# B&R Automation Studio project DuctLines (part 2)

### IoMap.iom - X20CP1584/IoMap.iom
```iecst
VAR_CONFIG
	Cyclic#2.::ProcessorJogFwd AT %IX."X20DI4653a".DigitalInput01;
	Cyclic#2.::ProcessorJogRev AT %IX."X20DI4653a".DigitalInput02;
	Cyclic#1.::EStopClear AT %IX."X20DI4653a".DigitalInput04;
	Cyclic#1.::ElectricDriveEnable AT %QX."X20CM8281".DigitalOutput01;
	Cyclic#1.::ActualDAC1 AT %QW."X20CM8281".AnalogOutput01;
	Cyclic#1.::ProcessorEncoderReset AT %QX."X20DC137A".Encoder01Reset;
	Cyclic#2.::HolePunchUp AT %IX."X20DI4653".DigitalInput01;
	Cyclic#1.ProcessorDriveReady AT %IX."X20CM8281".DigitalInput01;
	Cyclic#1.CoilLineHalt AT %IX."X20DI4653".DigitalInput03;
	Cyclic#2.::PowerOn AT %IX."X20DI4653a".DigitalInput03;
	Cyclic#1.CoilLineRun AT %IX."X20DI4653".DigitalInput02;
	Cyclic#1.CoilLineReset AT %IX."X20DI4653".DigitalInput04;
	Cyclic#2.::CoilLineRunIndicator AT %QX."X20DO6639".DigitalOutput01;
	Cyclic#2.::CoilLineHaltIndicator AT %QX."X20DO6639".DigitalOutput02;
	Cyclic#2.::ShearValve AT %QX."X20DO6639".DigitalOutput04;
	Cyclic#2.LTValve AT %QX."X20DO6639a".DigitalOutput01;
	Cyclic#2.VValve AT %QX."X20DO6639a".DigitalOutput02;
	Cyclic#2.LHoleValve AT %QX."X20DO6639a".DigitalOutput03;
	Cyclic#1.LevelerBrakeSolenoid AT %QX."X20DO6639a".DigitalOutput06;
	Cyclic#2.PunchMasterShiftSolenoid AT %QX."X20DO6639b".DigitalOutput01;
	Cyclic#2.OutSideGuideSolenoid AT %QX."X20DO6639b".DigitalOutput02;
	Cyclic#2.FourFootCenterSolenoid AT %QX."X20DO6639b".DigitalOutput03;
	Cyclic#2.FiveFootCenterSolenoid AT %QX."X20DO6639b".DigitalOutput04;
	Cyclic#2.SixFootCenterSolenoid AT %QX."X20DO6639b".DigitalOutput05;
	Cyclic#2.FourFootOutsideSolenoid AT %QX."X20DO6639b".DigitalOutput06;
	Cyclic#2.FiveFootOutsideSolenoid AT %QX."X20DO6639c".DigitalOutput01;
	Cyclic#2.SixFootOutsideSolenoid AT %QX."X20DO6639c".DigitalOutput02;
	Cyclic#2.DamperHoleSolenoid AT %QX."X20DO6639c".DigitalOutput03;
	Cyclic#2.HolePunchSelectedSolenoid AT %QX."X20DO6639c".DigitalOutput04;
	Cyclic#2.DieSelectSolenoid AT %QX."X20DO6639c".DigitalOutput05;
	Cyclic#1.::ActlMetalEncoder AT %ID."X20DC137A".Encoder01;
	Cyclic#2.BackGaugeJogInPB AT %IX."X20DI4653f".DigitalInput01;
	Cyclic#2.BackGaugeJogOutPB AT %IX."X20DI4653f".DigitalInput02;
	Cyclic#2.BackGaugeHomeLS AT %IX."X20DI4653f".DigitalInput03;
	Cyclic#2.FWBResetPB AT %IX."X20DI4653f".DigitalInput04;
	Cyclic#2.::PinspotEncoderResetSignal AT %QX."X20DC137A1".Encoder01Reset;
	Cyclic#2.BrakeEncoder AT %ID."X20DC137A2".Encoder01;
	Cyclic#2.BrakeEncoderReset AT %QX."X20DC137A2".Encoder01Reset;
	Cyclic#1.::ActualDAC2 AT %QW."X20CM8281a".AnalogOutput01;
	Cyclic#2.::BrakeDriveEnable AT %QX."X20CM8281a".DigitalOutput01;
	Cyclic#2.::BrakeDriveReset AT %QX."X20CM8281a".DigitalOutput02;
	Cyclic#2.::BrakeDriveReady AT %IX."X20CM8281a".DigitalInput01;
	Cyclic#1.::TSCEF1Button AT %IX."X20DI4653c".DigitalInput01;
	Cyclic#1.::TSCEF2Button AT %IX."X20DI4653c".DigitalInput02;
	Cyclic#1.::FullCleatSelect AT %IX."X20DI4653c".DigitalInput04;
	Cyclic#2.::PartPresentPSpotter AT %IX."X20DI4653d".DigitalInput04;
	Cyclic#2.::GuideSideStopLS AT %IX."X20DI4653g".DigitalInput01;
	Cyclic#2.::OperatorSideStopLS AT %IX."X20DI4653g".DigitalInput02;
	Cyclic#2.::BrakeAutoButton AT %IX."X20DI4653g".DigitalInput03;
	Cyclic#2.::BrakeHydraulicMS AT %IX."X20DI4653g".DigitalInput04;
	Cyclic#2.LatchCylinderInLS AT %IX."X20DI4653h".DigitalInput01;
	Cyclic#2.LatchCylinderOutLS AT %IX."X20DI4653h".DigitalInput02;
	Cyclic#2.::BrakeClampUpLS AT %IX."X20DI4653h".DigitalInput03;
	Cyclic#2.::BrakeClampDownLS AT %IX."X20DI4653i".DigitalInput01;
	Cyclic#2.::FormHeadUpLS AT %IX."X20DI4653i".DigitalInput02;
	Cyclic#2.::FormHeadDownLS AT %IX."X20DI4653i".DigitalInput03;
	Cyclic#2.::RotateStopsOut AT %IX."X20DI4653i".DigitalInput04;
	Cyclic#2.::RearEjectResetLimitSwitch AT %IX."X20DI4653j".DigitalInput01;
	Cyclic#2.::SmallPartsPusherLS AT %IX."X20DI4653j".DigitalInput04;
	Cyclic#2.::ManualClampPB AT %IX."X20DI4653j".DigitalInput03;
	Cyclic#1.SlowSpeedSolenoid AT %QX."X20DO6639".DigitalOutput03;
	Cyclic#1.::ForwardFeedSolenoid AT %QX."X20DO6639a".DigitalOutput04;
	Cyclic#1.::ReverseFeedSolenoid AT %QX."X20DO6639a".DigitalOutput05;
	Cyclic#2.::PinspotterDrive AT %QX."X20DO6639g".DigitalOutput01;
	Cyclic#2.::LatchCylinderInSolenoid AT %QX."X20DO6639i".DigitalOutput01;
	Cyclic#2.::LatchCylinderOutSolenoid AT %QX."X20DO6639i".DigitalOutput02;
	Cyclic#2.::BrakeBeamRaise AT %QX."X20DO6639i".DigitalOutput03;
	Cyclic#2.::BrakeBeamLower AT %QX."X20DO6639i".DigitalOutput04;
	Cyclic#2.::BrakeStopsInSolenoid AT %QX."X20DO6639j".DigitalOutput01;
	Cyclic#2.::BrakeStopsOutSolenoid AT %QX."X20DO6639j".DigitalOutput02;
	Cyclic#2.::SideEjectSolenoid AT %QX."X20DO6639j".DigitalOutput03;
	Cyclic#2.::FormHeadDownSolenoid AT %QX."X20DO6639j".DigitalOutput04;
	Cyclic#2.SmallPartPusherFwdSolenoid AT %QX."X20DO6639k".DigitalOutput01;
	Cyclic#2.SmallPartPusherRevSolenoid AT %QX."X20DO6639k".DigitalOutput02;
	Cyclic#2.FWBUnloaderValve AT %QX."X20DO6639k".DigitalOutput03;
	Cyclic#2.BrakeAutoIndicator AT %QX."X20DO6639k".DigitalOutput04;
	Cyclic#1.::CEF1Indicator AT %QX."X20DO6639d".DigitalOutput02;
	Cyclic#1.::CEF2Indicator AT %QX."X20DO6639d".DigitalOutput03;
	Cyclic#2.::FormHeadUpSolenoid AT %QX."X20DO6639i".DigitalOutput05;
	Cyclic#2.::SideEjectLiftSolenoid AT %QX."X20DO6639i".DigitalOutput06;
	Cyclic#1.::CEFNotchDetect AT %IX."X20DC137A".DigitalInput01;
	Cyclic#2.::PinspotEncoder AT %ID."X20DC137A1".Encoder01;
	Cyclic#2.::PinspotterLoad AT %QX."X20DO6639g".DigitalOutput03;
	Cyclic#2.::LinerAirSupply AT %QX."X20DO6639g".DigitalOutput05;
	Cyclic#2.DH800TOutPB AT %IX."X20DI4653b".DigitalInput01;
	Cyclic#2.DH800TInPB AT %IX."X20DI4653b".DigitalInput02;
	Cyclic#2.DH800TOutCR AT %QX."X20DO6639e".DigitalOutput01;
	Cyclic#2.DH800TInCR AT %QX."X20DO6639e".DigitalOutput02;
	Cyclic#2.DH800CEFOutCR AT %QX."X20DO6639d".DigitalOutput01;
	Cyclic#2.DH800CEFInCR AT %QX."X20DO6639d".DigitalOutput04;
	Cyclic#2.DH800CEFCalibrateCR AT %QX."X20DO6639d".DigitalOutput05;
	Cyclic#2.DH800CEFSlowCR AT %QX."X20DO6639d".DigitalOutput06;
	Cyclic#2.::DH800CEFInPB AT %IX."X20DI4653d".DigitalInput01;
	Cyclic#2.::DH800CEFOutPB AT %IX."X20DI4653d".DigitalInput03;
	Cyclic#1.BackGaugeAirBrake AT %QX."X20DO6639k".DigitalOutput05;
	Cyclic#2.::BrakePartEjectSolenoid AT %QX."X20DO6639j".DigitalOutput05;
END_VAR
```

## Configuration E1000V2_2

### Task classes (Cpu.sw)
```
Cyclic#1 (cycle 1000 us, tolerance 0 us):
  CEF <- CEF.prg
  IMotion2 <- IMotion2.prg
  EFdrHydDrv <- EFdrHydDrv1.prg
Cyclic#2 (cycle 20000 us, tolerance 20000 us):
  SysCheck <- SysCheck.prg
  E2Feeder <- E2Feeder.prg
  PMaster <- PMaster.prg
  Pinspotter <- Pinspotter.prg
  E_FWB <- E_FWB.prg
  DH800 <- DH800.prg
Cyclic#4 (cycle 100000 us, tolerance 100000 us):
  Server <- LibAsTCP1_ST.Server.prg
Binaries: sysconf, Role, User, iomap, ashwd, asfw, arconfig, TCData
Libraries: astcp, astime, standard, asieccon, runtime, asstring
```

### Hardware
same as Physical/E1000V2_1/Hardware.hw

### IoMap.iom - X20CP1584/IoMap.iom
```iecst
VAR_CONFIG
	Cyclic#2.::ProcessorJogFwd AT %IX."X20DI4653a".DigitalInput01;
	Cyclic#2.::ProcessorJogRev AT %IX."X20DI4653a".DigitalInput02;
	Cyclic#1.::EStopClear AT %IX."X20DI4653a".DigitalInput04;
	Cyclic#1.::ElectricDriveEnable AT %QX."X20CM8281".DigitalOutput01;
	Cyclic#1.::ActualDAC1 AT %QW."X20CM8281".AnalogOutput01;
	Cyclic#1.::ProcessorEncoderReset AT %QX."X20DC137A".Encoder01Reset;
	Cyclic#2.::HolePunchUp AT %IX."X20DI4653".DigitalInput01;
	Cyclic#1.ProcessorDriveReady AT %IX."X20CM8281".DigitalInput01;
	Cyclic#1.CoilLineHalt AT %IX."X20DI4653".DigitalInput03;
	Cyclic#2.::PowerOn AT %IX."X20DI4653a".DigitalInput03;
	Cyclic#1.CoilLineRun AT %IX."X20DI4653".DigitalInput02;
	Cyclic#1.CoilLineReset AT %IX."X20DI4653".DigitalInput04;
	Cyclic#2.::CoilLineRunIndicator AT %QX."X20DO6639".DigitalOutput01;
	Cyclic#2.::CoilLineHaltIndicator AT %QX."X20DO6639".DigitalOutput02;
	Cyclic#2.::ShearValve AT %QX."X20DO6639".DigitalOutput04;
	Cyclic#2.LTValve AT %QX."X20DO6639a".DigitalOutput01;
	Cyclic#2.VValve AT %QX."X20DO6639a".DigitalOutput02;
	Cyclic#2.LHoleValve AT %QX."X20DO6639a".DigitalOutput03;
	Cyclic#1.LevelerBrakeSolenoid AT %QX."X20DO6639a".DigitalOutput06;
	Cyclic#2.PunchMasterShiftSolenoid AT %QX."X20DO6639b".DigitalOutput01;
	Cyclic#2.OutSideGuideSolenoid AT %QX."X20DO6639b".DigitalOutput02;
	Cyclic#2.FourFootCenterSolenoid AT %QX."X20DO6639b".DigitalOutput03;
	Cyclic#2.FiveFootCenterSolenoid AT %QX."X20DO6639b".DigitalOutput04;
	Cyclic#2.SixFootCenterSolenoid AT %QX."X20DO6639b".DigitalOutput05;
	Cyclic#2.FourFootOutsideSolenoid AT %QX."X20DO6639b".DigitalOutput06;
	Cyclic#2.FiveFootOutsideSolenoid AT %QX."X20DO6639c".DigitalOutput01;
	Cyclic#2.SixFootOutsideSolenoid AT %QX."X20DO6639c".DigitalOutput02;
	Cyclic#2.DamperHoleSolenoid AT %QX."X20DO6639c".DigitalOutput03;
	Cyclic#2.HolePunchSelectedSolenoid AT %QX."X20DO6639c".DigitalOutput04;
	Cyclic#2.DieSelectSolenoid AT %QX."X20DO6639c".DigitalOutput05;
	Cyclic#1.::ActlMetalEncoder AT %ID."X20DC137A".Encoder01;
	Cyclic#2.BackGaugeJogInPB AT %IX."X20DI4653f".DigitalInput01;
	Cyclic#2.BackGaugeJogOutPB AT %IX."X20DI4653f".DigitalInput02;
	Cyclic#2.BackGaugeHomeLS AT %IX."X20DI4653f".DigitalInput03;
	Cyclic#2.FWBResetPB AT %IX."X20DI4653f".DigitalInput04;
	Cyclic#2.::PinspotEncoderResetSignal AT %QX."X20DC137A1".Encoder01Reset;
	Cyclic#2.BrakeEncoder AT %ID."X20DC137A2".Encoder01;
	Cyclic#2.BrakeEncoderReset AT %QX."X20DC137A2".Encoder01Reset;
	Cyclic#1.::ActualDAC2 AT %QW."X20CM8281a".AnalogOutput01;
	Cyclic#2.::BrakeDriveEnable AT %QX."X20CM8281a".DigitalOutput01;
	Cyclic#2.::BrakeDriveReset AT %QX."X20CM8281a".DigitalOutput02;
	Cyclic#2.::BrakeDriveReady AT %IX."X20CM8281a".DigitalInput01;
	Cyclic#1.::TSCEF1Button AT %IX."X20DI4653c".DigitalInput01;
	Cyclic#1.::TSCEF2Button AT %IX."X20DI4653c".DigitalInput02;
	Cyclic#1.::FullCleatSelect AT %IX."X20DI4653c".DigitalInput04;
	Cyclic#2.::PartPresentPSpotter AT %IX."X20DI4653d".DigitalInput04;
	Cyclic#2.::GuideSideStopLS AT %IX."X20DI4653g".DigitalInput01;
	Cyclic#2.::OperatorSideStopLS AT %IX."X20DI4653g".DigitalInput02;
	Cyclic#2.::BrakeAutoButton AT %IX."X20DI4653g".DigitalInput03;
	Cyclic#2.::BrakeHydraulicMS AT %IX."X20DI4653g".DigitalInput04;
	Cyclic#2.LatchCylinderInLS AT %IX."X20DI4653h".DigitalInput01;
	Cyclic#2.LatchCylinderOutLS AT %IX."X20DI4653h".DigitalInput02;
	Cyclic#2.::BrakeClampUpLS AT %IX."X20DI4653h".DigitalInput03;
	Cyclic#2.::BrakeClampDownLS AT %IX."X20DI4653i".DigitalInput01;
	Cyclic#2.::FormHeadUpLS AT %IX."X20DI4653i".DigitalInput02;
	Cyclic#2.::FormHeadDownLS AT %IX."X20DI4653i".DigitalInput03;
	Cyclic#2.::RotateStopsOut AT %IX."X20DI4653i".DigitalInput04;
	Cyclic#2.::RearEjectResetLimitSwitch AT %IX."X20DI4653j".DigitalInput01;
	Cyclic#2.::SmallPartsPusherLS AT %IX."X20DI4653j".DigitalInput04;
	Cyclic#2.::ManualClampPB AT %IX."X20DI4653j".DigitalInput03;
	Cyclic#1.SlowSpeedSolenoid AT %QX."X20DO6639".DigitalOutput03;
	Cyclic#1.::ForwardFeedSolenoid AT %QX."X20DO6639a".DigitalOutput04;
	Cyclic#1.::ReverseFeedSolenoid AT %QX."X20DO6639a".DigitalOutput05;
	Cyclic#2.::PinspotterDrive AT %QX."X20DO6639g".DigitalOutput01;
	Cyclic#2.::LatchCylinderInSolenoid AT %QX."X20DO6639i".DigitalOutput01;
	Cyclic#2.::LatchCylinderOutSolenoid AT %QX."X20DO6639i".DigitalOutput02;
	Cyclic#2.::BrakeBeamRaise AT %QX."X20DO6639i".DigitalOutput03;
	Cyclic#2.::BrakeBeamLower AT %QX."X20DO6639i".DigitalOutput04;
	Cyclic#2.::BrakeStopsInSolenoid AT %QX."X20DO6639j".DigitalOutput01;
	Cyclic#2.::BrakeStopsOutSolenoid AT %QX."X20DO6639j".DigitalOutput02;
	Cyclic#2.::SideEjectSolenoid AT %QX."X20DO6639j".DigitalOutput03;
	Cyclic#2.::FormHeadDownSolenoid AT %QX."X20DO6639j".DigitalOutput04;
	Cyclic#2.SmallPartPusherFwdSolenoid AT %QX."X20DO6639k".DigitalOutput01;
	Cyclic#2.SmallPartPusherRevSolenoid AT %QX."X20DO6639k".DigitalOutput02;
	Cyclic#2.FWBUnloaderValve AT %QX."X20DO6639k".DigitalOutput03;
	Cyclic#2.BrakeAutoIndicator AT %QX."X20DO6639k".DigitalOutput04;
	Cyclic#1.::CEF1Indicator AT %QX."X20DO6639d".DigitalOutput02;
	Cyclic#1.::CEF2Indicator AT %QX."X20DO6639d".DigitalOutput03;
	Cyclic#2.::FormHeadUpSolenoid AT %QX."X20DO6639i".DigitalOutput05;
	Cyclic#2.::SideEjectLiftSolenoid AT %QX."X20DO6639i".DigitalOutput06;
	Cyclic#1.::CEFNotchDetect AT %IX."X20DC137A".DigitalInput01;
	Cyclic#2.::PinspotEncoder AT %ID."X20DC137A1".Encoder01;
	Cyclic#2.::PinspotterLoad AT %QX."X20DO6639g".DigitalOutput03;
	Cyclic#2.::LinerAirSupply AT %QX."X20DO6639g".DigitalOutput05;
	Cyclic#2.DH800TOutPB AT %IX."X20DI4653b".DigitalInput01;
	Cyclic#2.DH800TInPB AT %IX."X20DI4653b".DigitalInput02;
	Cyclic#2.DH800TOutCR AT %QX."X20DO6639e".DigitalOutput01;
	Cyclic#2.DH800TInCR AT %QX."X20DO6639e".DigitalOutput02;
	Cyclic#2.DH800CEFOutCR AT %QX."X20DO6639d".DigitalOutput01;
	Cyclic#2.DH800CEFInCR AT %QX."X20DO6639d".DigitalOutput04;
	Cyclic#2.DH800CEFCalibrateCR AT %QX."X20DO6639d".DigitalOutput05;
	Cyclic#2.DH800CEFSlowCR AT %QX."X20DO6639d".DigitalOutput06;
	Cyclic#2.::DH800CEFInPB AT %IX."X20DI4653d".DigitalInput01;
	Cyclic#2.::DH800CEFOutPB AT %IX."X20DI4653d".DigitalInput03;
	Cyclic#1.BackGaugeAirBrake AT %QX."X20DO6639k".DigitalOutput05;
	Cyclic#2.::BrakePartEjectSolenoid AT %QX."X20DO6639j".DigitalOutput05;
	Cyclic#2.::DH800CEFCalibratePB AT %IX."X20DI4653d".DigitalInput02;
END_VAR
```

## Configuration E2000

CPU X20CP1584, AutomationRuntime J4.25, Build 4.1.2, Vc V4.25.0, Safety 0.0

### Hardware
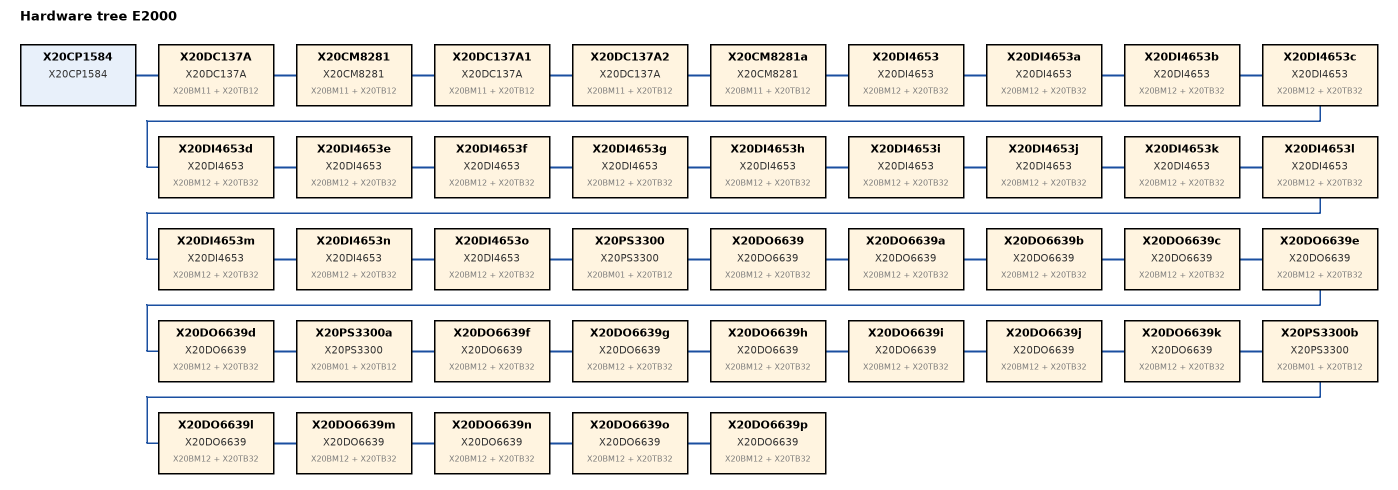
```
X20BM01 : X20BM01 v1.0.1.1  [X2X1 -> X20BM12aa.X2X2]
X20BM01a : X20BM01 v1.0.1.1  [X2X1 -> X20BM12o.X2X2]
X20BM01b : X20BM01 v1.0.1.1  [X2X1 -> X20BM12v.X2X2]
X20BM11 : X20BM11 v1.0.0.1  [X2X1 -> X20CP1584.IF6]
X20BM11a : X20BM11 v1.0.0.1  [X2X1 -> X20BM11.X2X2]
X20BM11b : X20BM11 v1.0.0.1  [X2X1 -> X20BM11a.X2X2]
X20BM11c : X20BM11 v1.0.0.1  [X2X1 -> X20BM11b.X2X2]
X20BM11d : X20BM11 v1.0.0.1  [X2X1 -> X20BM11c.X2X2]
X20BM12 : X20BM12 v1.0.0.1  [X2X1 -> X20BM11d.X2X2]
X20BM12a : X20BM12 v1.0.0.1  [X2X1 -> X20BM12.X2X2]
X20BM12aa : X20BM12 v1.0.0.1  [X2X1 -> X20BM12z.X2X2]
X20BM12ab : X20BM12 v1.0.0.1  [X2X1 -> X20BM01b.X2X2]
X20BM12ac : X20BM12 v1.0.0.1  [X2X1 -> X20BM12ab.X2X2]
X20BM12ad : X20BM12 v1.0.0.1  [X2X1 -> X20BM12ac.X2X2]
X20BM12ae : X20BM12 v1.0.0.1  [X2X1 -> X20BM12ad.X2X2]
X20BM12af : X20BM12 v1.0.0.1  [X2X1 -> X20BM12ae.X2X2]
X20BM12b : X20BM12 v1.0.0.1  [X2X1 -> X20BM12a.X2X2]
X20BM12c : X20BM12 v1.0.0.1  [X2X1 -> X20BM12b.X2X2]
X20BM12d : X20BM12 v1.0.0.1  [X2X1 -> X20BM12c.X2X2]
X20BM12e : X20BM12 v1.0.0.1  [X2X1 -> X20BM12d.X2X2]
X20BM12f : X20BM12 v1.0.0.1  [X2X1 -> X20BM12e.X2X2]
X20BM12g : X20BM12 v1.0.0.1  [X2X1 -> X20BM12f.X2X2]
X20BM12h : X20BM12 v1.0.0.1  [X2X1 -> X20BM12g.X2X2]
X20BM12i : X20BM12 v1.0.0.1  [X2X1 -> X20BM12h.X2X2]
X20BM12j : X20BM12 v1.0.0.1  [X2X1 -> X20BM12i.X2X2]
X20BM12k : X20BM12 v1.0.0.1  [X2X1 -> X20BM01.X2X2]
X20BM12l : X20BM12 v1.0.0.1  [X2X1 -> X20BM12k.X2X2]
X20BM12m : X20BM12 v1.0.0.1  [X2X1 -> X20BM12l.X2X2]
X20BM12n : X20BM12 v1.0.0.1  [X2X1 -> X20BM12m.X2X2]
X20BM12o : X20BM12 v1.0.0.1  [X2X1 -> X20BM12p.X2X2]
X20BM12p : X20BM12 v1.0.0.1  [X2X1 -> X20BM12n.X2X2]
X20BM12q : X20BM12 v1.0.0.1  [X2X1 -> X20BM01a.X2X2]
X20BM12r : X20BM12 v1.0.0.1  [X2X1 -> X20BM12q.X2X2]
X20BM12s : X20BM12 v1.0.0.1  [X2X1 -> X20BM12r.X2X2]
X20BM12t : X20BM12 v1.0.0.1  [X2X1 -> X20BM12s.X2X2]
X20BM12u : X20BM12 v1.0.0.1  [X2X1 -> X20BM12t.X2X2]
X20BM12v : X20BM12 v1.0.0.1  [X2X1 -> X20BM12u.X2X2]
X20BM12w : X20BM12 v1.0.0.1  [X2X1 -> X20BM12j.X2X2]
X20BM12x : X20BM12 v1.0.0.1  [X2X1 -> X20BM12w.X2X2]
X20BM12y : X20BM12 v1.0.0.1  [X2X1 -> X20BM12x.X2X2]
X20BM12z : X20BM12 v1.0.0.1  [X2X1 -> X20BM12y.X2X2]
X20CM8281 : X20CM8281 v1.0.4.0  [SS1 -> X20TB12a.SS; SL -> X20BM11a.SL1]
  Supervision = off
X20CM8281a : X20CM8281 v1.0.4.0  [SS1 -> X20TB12d.SS; SL -> X20BM11d.SL1]
  Supervision = off
X20CP1584 : X20CP1584 v1.3.0.0
  Connector IF2:
    ActivateDevice = 1
    EthInterfaceRedundant = 0
    Mode = Manual
    InternetAddress = 10.1.254.101
  Connector IF3:
    EplInterfaceRedundant = 0
    EplEthInterfaceRedundant = 0
  Connector IF6:
    CycleTime = 1000
  ConfigurationID = X20_CPU_E1000
  EnableUsbRemoteInstall = 1
  TimerDeviceType = EPLX2X
  TimerDevice = X20CP1584.IF6
  Cyclic1Duration = 1000
  Cyclic1Tolerance = 0
  Cyclic1Output = 1
  Cyclic2Duration = 20000
  Cyclic2Tolerance = 20000
  Cyclic3Duration = 50000
  Cyclic3Tolerance = 50000
  Cyclic4Duration = 100000
  Cyclic4Tolerance = 100000
  Cyclic5Duration = 200000
  Cyclic5Tolerance = 200000
  Cyclic6Duration = 500000
  Cyclic6Tolerance = 500000
  Cyclic7Duration = 1000000
  Cyclic7Tolerance = 1000000
  Cyclic8Duration = 10000
  Cyclic8Tolerance = 30000000
  Route1
X20DC137A : X20DC137A v1.0.0.3  [SS1 -> X20TB12.SS; SL -> X20BM11.SL1]
  Supervision = off
  CounterStd01 = 32Bit
  BWConfigChannel03 = off
X20DC137A1 : X20DC137A v1.0.0.3  [SS1 -> X20TB12b.SS; SL -> X20BM11b.SL1]
  Supervision = off
  CounterStd01 = 32Bit
  BWConfigChannel03 = off
X20DC137A2 : X20DC137A v1.0.0.3  [SS1 -> X20TB12c.SS; SL -> X20BM11c.SL1]
  Supervision = off
  CounterStd01 = 32Bit
  BWConfigChannel03 = off
X20DI4653 : X20DI4653 v1.0.2.0  [SS1 -> X20TB32.SS; SL -> X20BM12.SL1]
  Supervision = off
X20DI4653a : X20DI4653 v1.0.2.0  [SS1 -> X20TB32a.SS; SL -> X20BM12a.SL1]
  Supervision = off
X20DI4653b : X20DI4653 v1.0.2.0  [SS1 -> X20TB32b.SS; SL -> X20BM12b.SL1]
  Supervision = off
X20DI4653c : X20DI4653 v1.0.2.0  [SS1 -> X20TB32c.SS; SL -> X20BM12c.SL1]
  Supervision = off
X20DI4653d : X20DI4653 v1.0.2.0  [SS1 -> X20TB32d.SS; SL -> X20BM12d.SL1]
  Supervision = off
X20DI4653e : X20DI4653 v1.0.2.0  [SS1 -> X20TB32e.SS; SL -> X20BM12e.SL1]
  Supervision = off
X20DI4653f : X20DI4653 v1.0.2.0  [SS1 -> X20TB32f.SS; SL -> X20BM12f.SL1]
  Supervision = off
X20DI4653g : X20DI4653 v1.0.2.0  [SS1 -> X20TB32g.SS; SL -> X20BM12g.SL1]
  Supervision = off
X20DI4653h : X20DI4653 v1.0.2.0  [SS1 -> X20TB32h.SS; SL -> X20BM12h.SL1]
  Supervision = off
X20DI4653i : X20DI4653 v1.0.2.0  [SS1 -> X20TB32i.SS; SL -> X20BM12i.SL1]
  Supervision = off
X20DI4653j : X20DI4653 v1.0.2.0  [SS1 -> X20TB32j.SS; SL -> X20BM12j.SL1]
  Supervision = off
X20DI4653k : X20DI4653 v1.0.2.0  [SS1 -> X20TB32w.SS; SL -> X20BM12w.SL1]
  Supervision = off
X20DI4653l : X20DI4653 v1.0.2.0  [SS1 -> X20TB32x.SS; SL -> X20BM12x.SL1]
  Supervision = off
X20DI4653m : X20DI4653 v1.0.2.0  [SS1 -> X20TB32y.SS; SL -> X20BM12y.SL1]
  Supervision = off
X20DI4653n : X20DI4653 v1.0.2.0  [SS1 -> X20TB32z.SS; SL -> X20BM12z.SL1]
  Supervision = off
X20DI4653o : X20DI4653 v1.0.2.0  [SS1 -> X20TB32aa.SS; SL -> X20BM12aa.SL1]
  Supervision = off
X20DO6639 : X20DO6639 v1.0.1.0  [SS1 -> X20TB32k.SS; SL -> X20BM12k.SL1]
  Supervision = off
X20DO6639a : X20DO6639 v1.0.1.0  [SS1 -> X20TB32l.SS; SL -> X20BM12l.SL1]
  Supervision = off
X20DO6639b : X20DO6639 v1.0.1.0  [SS1 -> X20TB32m.SS; SL -> X20BM12m.SL1]
  Supervision = off
X20DO6639c : X20DO6639 v1.0.1.0  [SS1 -> X20TB32n.SS; SL -> X20BM12n.SL1]
  Supervision = off
X20DO6639d : X20DO6639 v1.0.1.0  [SS1 -> X20TB32o.SS; SL -> X20BM12o.SL1]
  Supervision = off
X20DO6639e : X20DO6639 v1.0.1.0  [SS1 -> X20TB32p.SS; SL -> X20BM12p.SL1]
  Supervision = off
X20DO6639f : X20DO6639 v1.0.1.0  [SS1 -> X20TB32q.SS; SL -> X20BM12q.SL1]
  Supervision = off
X20DO6639g : X20DO6639 v1.0.1.0  [SS1 -> X20TB32r.SS; SL -> X20BM12r.SL1]
  Supervision = off
X20DO6639h : X20DO6639 v1.0.1.0  [SS1 -> X20TB32s.SS; SL -> X20BM12s.SL1]
  Supervision = off
X20DO6639i : X20DO6639 v1.0.1.0  [SS1 -> X20TB32t.SS; SL -> X20BM12t.SL1]
  Supervision = off
X20DO6639j : X20DO6639 v1.0.1.0  [SS1 -> X20TB32u.SS; SL -> X20BM12u.SL1]
  Supervision = off
X20DO6639k : X20DO6639 v1.0.1.0  [SS1 -> X20TB32v.SS; SL -> X20BM12v.SL1]
  Supervision = off
X20DO6639l : X20DO6639 v1.0.1.0  [SS1 -> X20TB32ab.SS; SL -> X20BM12ab.SL1]
  Supervision = off
X20DO6639m : X20DO6639 v1.0.1.0  [SS1 -> X20TB32ac.SS; SL -> X20BM12ac.SL1]
  Supervision = off
X20DO6639n : X20DO6639 v1.0.1.0  [SS1 -> X20TB32ad.SS; SL -> X20BM12ad.SL1]
  Supervision = off
X20DO6639o : X20DO6639 v1.0.1.0  [SS1 -> X20TB32ae.SS; SL -> X20BM12ae.SL1]
  Supervision = off
X20DO6639p : X20DO6639 v1.0.1.0  [SS1 -> X20TB32af.SS; SL -> X20BM12af.SL1]
  Supervision = off
X20PS3300 : X20PS3300 v1.1.0.0  [SS1 -> X20TB12e.SS; SL -> X20BM01.SL1]
  Supervision = off
X20PS3300a : X20PS3300 v1.1.0.0  [SS1 -> X20TB12f.SS; SL -> X20BM01a.SL1]
  Supervision = off
X20PS3300b : X20PS3300 v1.1.0.0  [SS1 -> X20TB12g.SS; SL -> X20BM01b.SL1]
  Supervision = off
X20TB12 : X20TB12 v1.0.0.0
X20TB12a : X20TB12 v1.0.0.0
X20TB12b : X20TB12 v1.0.0.0
X20TB12c : X20TB12 v1.0.0.0
X20TB12d : X20TB12 v1.0.0.0
X20TB12e : X20TB12 v1.0.0.0
X20TB12f : X20TB12 v1.0.0.0
X20TB12g : X20TB12 v1.0.0.0
X20TB32 : X20TB32 v1.0.0.1
X20TB32a : X20TB32 v1.0.0.1
X20TB32aa : X20TB32 v1.0.0.1
X20TB32ab : X20TB32 v1.0.0.1
X20TB32ac : X20TB32 v1.0.0.1
X20TB32ad : X20TB32 v1.0.0.1
X20TB32ae : X20TB32 v1.0.0.1
X20TB32af : X20TB32 v1.0.0.1
X20TB32b : X20TB32 v1.0.0.1
X20TB32c : X20TB32 v1.0.0.1
X20TB32d : X20TB32 v1.0.0.1
X20TB32e : X20TB32 v1.0.0.1
X20TB32f : X20TB32 v1.0.0.1
X20TB32g : X20TB32 v1.0.0.1
X20TB32h : X20TB32 v1.0.0.1
X20TB32i : X20TB32 v1.0.0.1
X20TB32j : X20TB32 v1.0.0.1
X20TB32k : X20TB32 v1.0.0.1
X20TB32l : X20TB32 v1.0.0.1
X20TB32m : X20TB32 v1.0.0.1
X20TB32n : X20TB32 v1.0.0.1
X20TB32o : X20TB32 v1.0.0.1
X20TB32p : X20TB32 v1.0.0.1
X20TB32q : X20TB32 v1.0.0.1
X20TB32r : X20TB32 v1.0.0.1
X20TB32s : X20TB32 v1.0.0.1
X20TB32t : X20TB32 v1.0.0.1
X20TB32u : X20TB32 v1.0.0.1
X20TB32v : X20TB32 v1.0.0.1
X20TB32w : X20TB32 v1.0.0.1
X20TB32x : X20TB32 v1.0.0.1
X20TB32y : X20TB32 v1.0.0.1
X20TB32z : X20TB32 v1.0.0.1
```

### IoMap.iom - X20CP1584/IoMap.iom
```iecst
VAR_CONFIG
	Cyclic#2.Uncoiler4Select AT %IX."X20DI4653a".DigitalInput02;
	Cyclic#2.Uncoiler6Select AT %IX."X20DI4653a".DigitalInput04;
	Cyclic#1.::ElectricDriveEnable AT %QX."X20CM8281".DigitalOutput01;
	Cyclic#1.::ActualDAC1 AT %QW."X20CM8281".AnalogOutput01;
	Cyclic#1.::ProcessorEncoderReset AT %QX."X20DC137A".Encoder01Reset;
	Cyclic#2.ProcessorDriveReady AT %IX."X20CM8281".DigitalInput01;
	Cyclic#2.Uncoiler5Select AT %IX."X20DI4653a".DigitalInput03;
	Cyclic#2.::Station1ForwardSolenoid AT %QX."X20DO6639".DigitalOutput04;
	Cyclic#2.Station2ForwardSolenoid AT %QX."X20DO6639a".DigitalOutput01;
	Cyclic#2.Station2ReverseSolenoid AT %QX."X20DO6639a".DigitalOutput02;
	Cyclic#2.Station2BrakeSolenoid AT %QX."X20DO6639a".DigitalOutput03;
	Cyclic#2.Station3BrakeSolenoid AT %QX."X20DO6639a".DigitalOutput06;
	Cyclic#2.Station4ForwardSolenoid AT %QX."X20DO6639b".DigitalOutput01;
	Cyclic#2.Station4ReverseSolenoid AT %QX."X20DO6639b".DigitalOutput02;
	Cyclic#2.Station4BrakeSolenoid AT %QX."X20DO6639b".DigitalOutput03;
	Cyclic#2.Station5ForwardSolenoid AT %QX."X20DO6639b".DigitalOutput04;
	Cyclic#2.Station5ReverseSolenoid AT %QX."X20DO6639b".DigitalOutput05;
	Cyclic#2.Station5BrakeSolenoid AT %QX."X20DO6639b".DigitalOutput06;
	Cyclic#2.Station6ForwardSolenoid AT %QX."X20DO6639c".DigitalOutput01;
	Cyclic#2.Station6ReverseSolenoid AT %QX."X20DO6639c".DigitalOutput02;
	Cyclic#2.Station6BrakeSolenoid AT %QX."X20DO6639c".DigitalOutput03;
	Cyclic#1.::ActlMetalEncoder AT %ID."X20DC137A".Encoder01;
	Cyclic#2.PinspotEncoder AT %ID."X20DC137A1".Encoder01;
	Cyclic#2.PinspotEncoderResetSignal AT %QX."X20DC137A1".Encoder01Reset;
	Cyclic#1.BrakeEncoder AT %ID."X20DC137A2".Encoder01;
	Cyclic#1.BrakeDriveEnable AT %QX."X20CM8281a".DigitalOutput01;
	Cyclic#1.BrakeDriveReset AT %QX."X20CM8281a".DigitalOutput02;
	Cyclic#2.BrakeDriveReady AT %IX."X20CM8281a".DigitalInput01;
	Cyclic#2.UncoilerAutoSwitch AT %IX."X20DI4653".DigitalInput01;
	Cyclic#2.UncoilerJogPB AT %IX."X20DI4653".DigitalInput02;
	Cyclic#2.Uncoiler1Select AT %IX."X20DI4653".DigitalInput03;
	Cyclic#2.Uncoiler2Select AT %IX."X20DI4653".DigitalInput04;
	Cyclic#2.Uncoiler3Select AT %IX."X20DI4653a".DigitalInput01;
	Cyclic#2.UncoilerStationLimitSwitch1 AT %IX."X20DI4653b".DigitalInput01;
	Cyclic#2.UncoilerStationLimitSwitch2 AT %IX."X20DI4653b".DigitalInput02;
	Cyclic#2.UncoilerStationLimitSwitch3 AT %IX."X20DI4653b".DigitalInput03;
	Cyclic#2.UncoilerStationLimitSwitch4 AT %IX."X20DI4653b".DigitalInput04;
	Cyclic#2.UncoilerStationLimitSwitch5 AT %IX."X20DI4653c".DigitalInput01;
	Cyclic#2.UncoilerStationLimitSwitch6 AT %IX."X20DI4653c".DigitalInput02;
	Cyclic#2.UncoilerRewindSwitch AT %IX."X20DI4653c".DigitalInput03;
	Cyclic#2.UncoilerUnwindSwitch AT %IX."X20DI4653c".DigitalInput04;
	Cyclic#2.HolePunchUp AT %IX."X20DI4653d".DigitalInput01;
	Cyclic#2.::ProcessorJogFwd AT %IX."X20DI4653d".DigitalInput02;
	Cyclic#2.::ProcessorJogRev AT %IX."X20DI4653d".DigitalInput03;
	Cyclic#1.PowerOn AT %IX."X20DI4653e".DigitalInput02;
	Cyclic#1.EStopClear AT %IX."X20DI4653e".DigitalInput04;
	Cyclic#2.HeadInPositionLS AT %IX."X20DI4653f".DigitalInput01;
	Cyclic#2.Pusher1OffProx AT %IX."X20DI4653f".DigitalInput02;
	Cyclic#2.Pusher2OffProx AT %IX."X20DI4653f".DigitalInput03;
	Cyclic#2.Table1SheetStopProxA AT %IX."X20DI4653f".DigitalInput04;
	Cyclic#2.Table1SheetStopProxB AT %IX."X20DI4653g".DigitalInput01;
	Cyclic#2.Table2SheetStopProxA AT %IX."X20DI4653g".DigitalInput02;
	Cyclic#2.Table2SheetStopProxB AT %IX."X20DI4653g".DigitalInput03;
	Cyclic#2.Lift3DownProx AT %IX."X20DI4653g".DigitalInput04;
	Cyclic#2.BypassSwitch AT %IX."X20DI4653h".DigitalInput01;
	Cyclic#2.Table1SideBypassLS AT %IX."X20DI4653h".DigitalInput02;
	Cyclic#2.CEFJogPB AT %IX."X20DI4653h".DigitalInput04;
	Cyclic#2.TDFJogPB AT %IX."X20DI4653i".DigitalInput01;
	Cyclic#2.LOMSpeedSelect1 AT %IX."X20DI4653i".DigitalInput02;
	Cyclic#2.LOMSpeedSelect2 AT %IX."X20DI4653i".DigitalInput03;
	Cyclic#2.::PartPresentPSpotter AT %IX."X20DI4653i".DigitalInput04;
	Cyclic#2.GuideSideStopLS AT %IX."X20DI4653j".DigitalInput01;
	Cyclic#2.OperatorSideStopLS AT %IX."X20DI4653j".DigitalInput02;
	Cyclic#2.BrakeClampUpLS AT %IX."X20DI4653j".DigitalInput03;
	Cyclic#2.BrakeClampMidwayLS AT %IX."X20DI4653j".DigitalInput04;
	Cyclic#2.BrakeClampDownLS AT %IX."X20DI4653k".DigitalInput01;
	Cyclic#2.FormHeadUpLS AT %IX."X20DI4653k".DigitalInput02;
	Cyclic#2.FormHeadDownLS AT %IX."X20DI4653k".DigitalInput03;
	Cyclic#2.RearEjectResetLimitSwitch AT %IX."X20DI4653k".DigitalInput04;
	Cyclic#2.BackGaugeHomeLS AT %IX."X20DI4653l".DigitalInput01;
	Cyclic#2.ManualClampPB AT %IX."X20DI4653l".DigitalInput02;
	Cyclic#2.SmallPartsPusherLS AT %IX."X20DI4653l".DigitalInput03;
	Cyclic#2.BackGaugeJogInPB AT %IX."X20DI4653l".DigitalInput04;
	Cyclic#2.BackGaugeJogOutPB AT %IX."X20DI4653m".DigitalInput01;
	Cyclic#2.SmallPartPusherHomeLS AT %IX."X20DI4653m".DigitalInput02;
	Cyclic#2.PartEjectHomeLS AT %IX."X20DI4653m".DigitalInput03;
	Cyclic#2.TripIndicatorCradles2 AT %IX."X20DI4653n".DigitalInput01;
	Cyclic#2.TripIndicatorCoilLine AT %IX."X20DI4653n".DigitalInput02;
	Cyclic#2.TripIndicatorTransfer1 AT %IX."X20DI4653n".DigitalInput03;
	Cyclic#2.TripIndicatorTransfer2 AT %IX."X20DI4653n".DigitalInput04;
	TripIndicatorCEF AT %IX."X20DI4653o".DigitalInput01;
	TripIndicatorTDF AT %IX."X20DI4653o".DigitalInput02;
	TripIndicatorPump AT %IX."X20DI4653o".DigitalInput03;
	Cyclic#2.BrakeHydraulics AT %IX."X20DI4653o".DigitalInput04;
	Cyclic#2.::Station1ReverseSolenoid AT %QX."X20DO6639".DigitalOutput05;
	Cyclic#2.::Station1BrakeSolenoid AT %QX."X20DO6639".DigitalOutput06;
	Cyclic#2.Statrion3ForwardSolenoid AT %QX."X20DO6639a".DigitalOutput04;
	Cyclic#2.Station3ReverseSolenoid AT %QX."X20DO6639a".DigitalOutput05;
	Cyclic#2.::FourFootCenterSolenoid AT %QX."X20DO6639e".DigitalOutput02;
	Cyclic#2.::LHoleValve AT %QX."X20DO6639e".DigitalOutput01;
	Cyclic#2.FiveFootCenterSolenoid AT %QX."X20DO6639e".DigitalOutput03;
	Cyclic#2.SixFootCenterSolenoid AT %QX."X20DO6639e".DigitalOutput04;
	Cyclic#2.::FourFootOutsideSolenoid AT %QX."X20DO6639d".DigitalOutput01;
	Cyclic#2.::FiveFootOutsideSolenoid AT %QX."X20DO6639d".DigitalOutput02;
	Cyclic#2.::SixFootOutsideSolenoid AT %QX."X20DO6639d".DigitalOutput03;
	Cyclic#2.::OutSideGuideSolenoid AT %QX."X20DO6639d".DigitalOutput04;
	Cyclic#2.::PunchMasterShiftSolenoid AT %QX."X20DO6639f".DigitalOutput01;
	Cyclic#2.DamperHoleSolenoid AT %QX."X20DO6639f".DigitalOutput02;
	Cyclic#1.SlowSpeedSolenoid AT %QX."X20DO6639f".DigitalOutput03;
	Cyclic#1.ForwardFeedSolenoid AT %QX."X20DO6639f".DigitalOutput04;
	Cyclic#1.ReverseFeedSolenoid AT %QX."X20DO6639f".DigitalOutput05;
	Cyclic#1.LevelerBrakeSolenoid AT %QX."X20DO6639f".DigitalOutput06;
	Cyclic#2.::ShearValve AT %QX."X20DO6639g".DigitalOutput01;
	Cyclic#2.::LTValve AT %QX."X20DO6639g".DigitalOutput02;
	Cyclic#2.::VValve AT %QX."X20DO6639g".DigitalOutput03;
	Cyclic#2.CoilLinePower AT %QX."X20DO6639g".DigitalOutput04;
	Cyclic#2.EZPunchSolenoid AT %QX."X20DO6639g".DigitalOutput05;
	Cyclic#2.Transfer1Power AT %QX."X20DO6639h".DigitalOutput01;
	Cyclic#2.Transfer2Power AT %QX."X20DO6639h".DigitalOutput02;
	Cyclic#2.Lift1Solenoid AT %QX."X20DO6639h".DigitalOutput03;
	Cyclic#2.Lift2Solenoid AT %QX."X20DO6639h".DigitalOutput04;
	Cyclic#2.Lift3UpSolenoid AT %QX."X20DO6639i".DigitalOutput01;
	Cyclic#2.Lift3DownSolenoid AT %QX."X20DO6639i".DigitalOutput02;
	Cyclic#2.Pusher1Solenoid AT %QX."X20DO6639i".DigitalOutput03;
	Cyclic#2.Pusher2Solenoid AT %QX."X20DO6639i".DigitalOutput04;
	Cyclic#1.StatHeadRollSolenoid AT %QX."X20DO6639j".DigitalOutput01;
	Cyclic#1.MoveHeadRollSolenoid AT %QX."X20DO6639j".DigitalOutput02;
	Cyclic#2.CEFPower AT %QX."X20DO6639j".DigitalOutput03;
	TDFPower AT %QX."X20DO6639k".DigitalOutput01;
	Cyclic#2.LOMLowSpeedRelay AT %QX."X20DO6639l".DigitalOutput01;
	Cyclic#2.LOMHiSpeedRelay AT %QX."X20DO6639l".DigitalOutput02;
	Cyclic#2.BrakeLowSpeedRelay AT %QX."X20DO6639l".DigitalOutput03;
	Cyclic#2.BrakeHiSpeedRelay AT %QX."X20DO6639l".DigitalOutput04;
	Cyclic#2.::PinspotterDrive AT %QX."X20DO6639m".DigitalOutput01;
	Cyclic#2.LOMConveyorRunRelay AT %QX."X20DO6639m".DigitalOutput02;
	Cyclic#2.::PinspotterLoad AT %QX."X20DO6639m".DigitalOutput03;
	Cyclic#2.LinerAirSupply AT %QX."X20DO6639m".DigitalOutput04;
	Cyclic#2.BrakeHydraulicMS AT %QX."X20DO6639n".DigitalOutput01;
	Cyclic#2.BrakeOutfeedConveyorMotor AT %QX."X20DO6639n".DigitalOutput02;
	Cyclic#2.::BrakeBeamRaise AT %QX."X20DO6639n".DigitalOutput03;
	Cyclic#2.::BrakeBeamLower AT %QX."X20DO6639n".DigitalOutput04;
	Cyclic#2.FormHeadUpSolenoid AT %QX."X20DO6639o".DigitalOutput01;
	Cyclic#2.BrakeStopsInSolenoid AT %QX."X20DO6639o".DigitalOutput02;
	Cyclic#2.BrakeStopsOutSolenoid AT %QX."X20DO6639o".DigitalOutput03;
	Cyclic#2.BrakePartEjectSolenoid AT %QX."X20DO6639o".DigitalOutput04;
	Cyclic#2.SmallPartPusherFwdSolenoid AT %QX."X20DO6639p".DigitalOutput01;
	Cyclic#2.SmallPartPusherRevSolenoid AT %QX."X20DO6639p".DigitalOutput02;
	Cyclic#1.BackGaugeAirBrake AT %QX."X20DO6639p".DigitalOutput03;
	Cyclic#2.BrakeInfeedConveyorMotor AT %QX."X20DO6639p".DigitalOutput04;
	Cyclic#2.::BrakeEncoderReset AT %QX."X20DC137A2".Encoder01Reset;
	Cyclic#2.CDADecoilPower AT %QX."X20DO6639".DigitalOutput01;
	Cyclic#1.::CEFNotchDetect AT %IX."X20DC137A".DigitalInput01;
	Cyclic#1.::ActualDAC2 AT %QW."X20CM8281a".AnalogOutput01;
END_VAR
```

## Configuration Southwark_CD2505_00

### Task classes (Cpu.sw)
```
Cyclic#1 (cycle 1000 us, tolerance 10000 us):
  IMotionCon <- IMotionControl.prg
  CleatRoll <- CleatRoll.prg
Cyclic#2 (cycle 10000 us, tolerance 20000 us):
  Uncoiler_1 <- Uncoiler_1.prg
  MarkTable <- MarkTable.prg
  MarkRF <- MarkRF.prg
  Feeder <- Feeder.prg
  SBrake <- SBrake.prg
  Pivot_2 <- Pivot_2.prg
  TDCTable <- TDCTable.prg
  TDCRFPshrs <- TDCRFPshrs.prg
  GlueApp <- GlueApp.prg
  Insulmatic <- Insulmatic.prg
  Pinspotter <- Pinspotter.prg
  BrakeCommo <- BrakeCommon.prg
  HydraulicB <- HydraulicBrakeCarriage.prg
  HWBwoPLC <- HWBwoPLC.prg
Cyclic#4 (cycle 100000 us, tolerance 100000 us):
  HMIButtons <- HMIButtons.prg
  Server <- LibAsTCP1_ST.Server.prg
Binaries: TCData, arconfig, asfw, ashwd, iomap, User, Role, sysconf
Libraries: standard, MestekLib, AsTCP, runtime, asstring, asieccon, astime
```

### Hardware
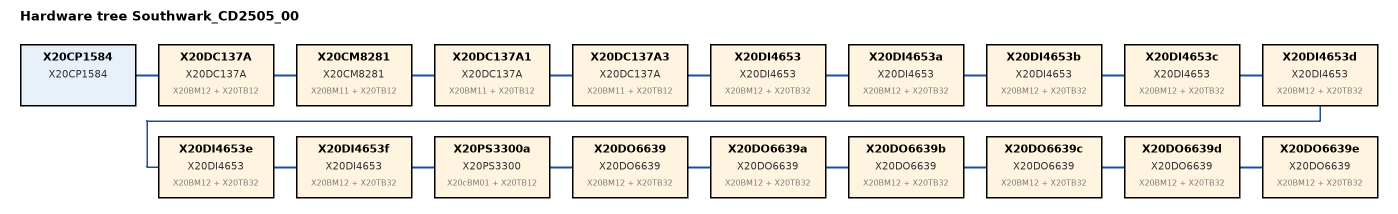
```
X20BM11 : X20BM11 v1.0.0.1  [X2X1 -> X20BM12a.X2X2]
X20BM11b : X20BM11 v1.0.0.1  [X2X1 -> X20BM11.X2X2]
X20BM11c : X20BM11 v1.0.0.1  [X2X1 -> X20BM11b.X2X2]
X20BM12 : X20BM12 v1.0.0.1  [X2X1 -> X20BM11c.X2X2]
X20BM12a : X20BM12 v1.0.0.1  [X2X1 -> X20CP1584.IF6]
X20BM12aa : X20BM12 v1.0.0.1  [X2X1 -> X20BM12z.X2X2]
X20BM12b : X20BM12 v1.0.0.1  [X2X1 -> X20BM12.X2X2]
X20BM12c : X20BM12 v1.0.0.1  [X2X1 -> X20BM12b.X2X2]
X20BM12d : X20BM12 v1.0.0.1  [X2X1 -> X20BM12c.X2X2]
X20BM12e : X20BM12 v1.0.0.1  [X2X1 -> X20BM12d.X2X2]
X20BM12f : X20BM12 v1.0.0.1  [X2X1 -> X20BM12e.X2X2]
X20BM12g : X20BM12 v1.0.0.1  [X2X1 -> X20BM12f.X2X2]
X20BM12v : X20BM12 v1.0.0.1  [X2X1 -> X20cBM01.X2X2]
X20BM12w : X20BM12 v1.0.0.1  [X2X1 -> X20BM12v.X2X2]
X20BM12x : X20BM12 v1.0.0.1  [X2X1 -> X20BM12w.X2X2]
X20BM12y : X20BM12 v1.0.0.1  [X2X1 -> X20BM12x.X2X2]
X20BM12z : X20BM12 v1.0.0.1  [X2X1 -> X20BM12y.X2X2]
X20CM8281 : X20CM8281 v1.0.4.0  [SS1 -> X20TB12.SS; SL -> X20BM11.SL1]
  Supervision = off
X20CP1584 : X20CP1584 v1.3.0.0
  Connector IF2:
    ActivateDevice = 1
    EthInterfaceRedundant = 0
    Mode = Manual
    InternetAddress = 10.1.254.101
  Connector IF3:
    EplInterfaceRedundant = 0
    EplEthInterfaceRedundant = 0
  ConfigurationID = X20_CPU_test
  EnableUsbRemoteInstall = 1
  TimerDeviceType = SWIOTIMER
  Cyclic1Duration = 1000
  Cyclic1Tolerance = 10000
  Cyclic2Duration = 10000
  Cyclic2Tolerance = 20000
  Cyclic3Duration = 50000
  Cyclic3Tolerance = 50000
  Cyclic4Duration = 100000
  Cyclic4Tolerance = 100000
  Cyclic5Duration = 200000
  Cyclic5Tolerance = 200000
  Cyclic6Duration = 500000
  Cyclic6Tolerance = 500000
  Cyclic7Duration = 1000000
  Cyclic7Tolerance = 1000000
  Cyclic8Duration = 10000
  Cyclic8Tolerance = 30000000
X20DC137A : X20DC137A v1.0.0.3  [SS1 -> X20TB12b.SS; SL -> X20BM12a.SL1]
  Supervision = off
  CounterStd01 = 32Bit
  BWConfigChannel03 = off
X20DC137A1 : X20DC137A v1.0.0.3  [SS1 -> X20TB12c.SS; SL -> X20BM11b.SL1]
  Supervision = off
  CounterStd01 = 32Bit
  BWConfigChannel03 = off
X20DC137A3 : X20DC137A v1.0.0.3  [SS1 -> X20TB12d.SS; SL -> X20BM11c.SL1]
  Supervision = off
  CounterStd01 = 32Bit
  BWConfigChannel03 = off
X20DI4653 : X20DI4653 v1.0.2.0  [SS1 -> X20TB32.SS; SL -> X20BM12.SL1]
  Supervision = off
X20DI4653a : X20DI4653 v1.0.2.0  [SS1 -> X20TB32a.SS; SL -> X20BM12b.SL1]
  Supervision = off
X20DI4653b : X20DI4653 v1.0.2.0  [SS1 -> X20TB32b.SS; SL -> X20BM12c.SL1]
  Supervision = off
X20DI4653c : X20DI4653 v1.0.2.0  [SS1 -> X20TB32c.SS; SL -> X20BM12d.SL1]
  Supervision = off
X20DI4653d : X20DI4653 v1.0.2.0  [SS1 -> X20TB32d.SS; SL -> X20BM12e.SL1]
  Supervision = off
X20DI4653e : X20DI4653 v1.0.2.0  [SS1 -> X20TB32e.SS; SL -> X20BM12f.SL1]
  Supervision = off
X20DI4653f : X20DI4653 v1.0.2.0  [SS1 -> X20TB32f.SS; SL -> X20BM12g.SL1]
  Supervision = off
X20DO6639 : X20DO6639 v1.0.1.0  [SS1 -> X20TB32u.SS; SL -> X20BM12v.SL1]
  Supervision = off
X20DO6639a : X20DO6639 v1.0.1.0  [SS1 -> X20TB32v.SS; SL -> X20BM12w.SL1]
  Supervision = off
X20DO6639b : X20DO6639 v1.0.1.0  [SS1 -> X20TB32w.SS; SL -> X20BM12x.SL1]
  Supervision = off
X20DO6639c : X20DO6639 v1.0.1.0  [SS1 -> X20TB32x.SS; SL -> X20BM12y.SL1]
  Supervision = off
X20DO6639d : X20DO6639 v1.0.1.0  [SS1 -> X20TB32y.SS; SL -> X20BM12z.SL1]
  Supervision = off
X20DO6639e : X20DO6639 v1.0.1.0  [SS1 -> X20TB32z.SS; SL -> X20BM12aa.SL1]
  Supervision = off
X20PS3300a : X20PS3300 v1.1.0.0  [SS1 -> X20TB12f.SS; SL -> X20cBM01.SL1]
  Supervision = off
X20TB12 : X20TB12 v1.0.0.0
X20TB12b : X20TB12 v1.0.0.0
X20TB12c : X20TB12 v1.0.0.0
X20TB12d : X20TB12 v1.0.0.0
X20TB12f : X20TB12 v1.0.0.0
X20TB32 : X20TB32 v1.0.0.1
X20TB32a : X20TB32 v1.0.0.1
X20TB32b : X20TB32 v1.0.0.1
X20TB32c : X20TB32 v1.0.0.1
X20TB32d : X20TB32 v1.0.0.1
X20TB32e : X20TB32 v1.0.0.1
X20TB32f : X20TB32 v1.0.0.1
X20TB32u : X20TB32 v1.0.0.1
X20TB32v : X20TB32 v1.0.0.1
X20TB32w : X20TB32 v1.0.0.1
X20TB32x : X20TB32 v1.0.0.1
X20TB32y : X20TB32 v1.0.0.1
X20TB32z : X20TB32 v1.0.0.1
X20cBM01 : X20cBM01 v1.0.1.0  [X2X1 -> X20BM12g.X2X2]
```

### IoMap.iom - X20CP1584/IoMap.iom
```iecst
VAR_CONFIG
	Cyclic#1.ActlMetalEncoder AT %ID."X20DC137A".Encoder01;
	Cyclic#1.::ProcessorEncoderReset AT %QX."X20DC137A".Encoder01Reset;
	Cyclic#1.ActualDAC1 AT %QW."X20CM8281".AnalogOutput01;
	Cyclic#1.ElectricDriveEnable AT %QX."X20CM8281".DigitalOutput01;
	Cyclic#2.MarkEncoderResetSignal AT %QX."X20DC137A1".Encoder01Reset;
	Cyclic#2.RawMarkEncoder AT %ID."X20DC137A1".Encoder01;
	Cyclic#2.::BrakeEncoderReset AT %QX."X20DC137A3".Encoder01Reset;
	Cyclic#2.BrakeEncoder AT %ID."X20DC137A3".Encoder01;
	Cyclic#2.EStopClear AT %IX."X20DI4653".DigitalInput01;
	Cyclic#2.FeedInitButton AT %IX."X20DI4653".DigitalInput04;
	Cyclic#2.ProcessorDriveEnable AT %IX."X20DI4653".DigitalInput03;
	Cyclic#2.UncoilerOnLatch AT %IX."X20DI4653".DigitalInput02;
	Cyclic#2.DuctoAuto AT %IX."X20DI4653a".DigitalInput01;
	Cyclic#2.MatlAtMeasureRoll AT %IX."X20DI4653a".DigitalInput04;
	Cyclic#2.ProcessorJogFwd AT %IX."X20DI4653a".DigitalInput02;
	Cyclic#2.ProcessorJogRev AT %IX."X20DI4653a".DigitalInput03;
	Cyclic#2.RotatingTableOn AT %IX."X20DI4653b".DigitalInput01;
	Cyclic#2.PartPresentRTClamp AT %IX."X20DI4653b".DigitalInput02;
	Cyclic#2.PartPresentRTKnurledRoll AT %IX."X20DI4653b".DigitalInput03;
	Cyclic#2.PartRotateComplete AT %IX."X20DI4653b".DigitalInput04;
	Cyclic#2.HumpLimitSwitch AT %IX."X20DI4653c".DigitalInput01;
	Cyclic#2.PowerOn AT %IX."X20DI4653c".DigitalInput04;
	Cyclic#2.SlackBar AT %IX."X20DI4653c".DigitalInput02;
	Cyclic#2.MarkAuto AT %IX."X20DI4653d".DigitalInput02;
	Cyclic#2.MarkRollformerOn AT %IX."X20DI4653d".DigitalInput01;
	Cyclic#2.MarkSetButton AT %IX."X20DI4653d".DigitalInput03;
	Cyclic#2.::MarkRefSwitch AT %IX."X20DI4653e".DigitalInput01;
	Cyclic#2.MarkHeadJogInSwitch AT %IX."X20DI4653e".DigitalInput03;
	Cyclic#2.MarkHeadJogOutSwitch AT %IX."X20DI4653e".DigitalInput04;
	Cyclic#2.MarkHiSpeedSignal AT %IX."X20DI4653e".DigitalInput02;
	Cyclic#2.::CarriageReference AT %IX."X20DI4653f".DigitalInput01;
	Cyclic#2.::BrakeAutoRequest AT %IX."X20DI4653f".DigitalInput03;
	Cyclic#2.AmberLight AT %QX."X20DO6639".DigitalOutput02;
	Cyclic#2.BatchActivePhysical AT %QX."X20DO6639".DigitalOutput06;
	Cyclic#2.BlockingValve AT %QX."X20DO6639".DigitalOutput05;
	Cyclic#2.BlueLight AT %QX."X20DO6639".DigitalOutput03;
	Cyclic#2.UncoilerRun AT %QX."X20DO6639".DigitalOutput04;
	Cyclic#2.WarningHorn AT %QX."X20DO6639".DigitalOutput01;
	Cyclic#2.LTValve AT %QX."X20DO6639a".DigitalOutput04;
	Cyclic#2.::CustomVValve AT %QX."X20DO6639a".DigitalOutput06;
	Cyclic#2.::CustomLTValve AT %QX."X20DO6639a".DigitalOutput05;
	Cyclic#2.ShearValve AT %QX."X20DO6639a".DigitalOutput01;
	Cyclic#2.SnapLockButtonGag AT %QX."X20DO6639a".DigitalOutput02;
	Cyclic#2.VValve AT %QX."X20DO6639a".DigitalOutput03;
	Cyclic#2.RTSkewTableRelay AT %QX."X20DO6639b".DigitalOutput01;
	Cyclic#2.RTBeltConveyorMotor AT %QX."X20DO6639b".DigitalOutput02;
	Cyclic#2.RTKnurledRollsMotor AT %QX."X20DO6639b".DigitalOutput03;
	Cyclic#2.RTBeltConveyorRaiseSolenoid AT %QX."X20DO6639b".DigitalOutput04;
	Cyclic#2.PivotClampCloseSolenoid AT %QX."X20DO6639b".DigitalOutput05;
	Cyclic#2.CushionRollRaiseSolenoid AT %QX."X20DO6639b".DigitalOutput06;
	Cyclic#2.RTPivotArmRotate AT %QX."X20DO6639c".DigitalOutput03;
	Cyclic#2.RTKnurledRollLowerSolenoid AT %QX."X20DO6639c".DigitalOutput01;
	Cyclic#2.RTKnurledRollGateSolenoid AT %QX."X20DO6639c".DigitalOutput02;
	Cyclic#2.::MarkRFHighSpeed AT %QX."X20DO6639d".DigitalOutput03;
	Cyclic#2.::BrakeHighSpeedRelay AT %QX."X20DO6639e".DigitalOutput03;
	Cyclic#2.::BrakeOn AT %QX."X20DO6639e".DigitalOutput04;
	::PartPresentMarkExit AT %IX."X20DI4653c".DigitalInput03;
	Cyclic#2.SmallPittsSelected AT %IX."X20DI4653d".DigitalInput04;
	Cyclic#2.::MarkRFMoveIn AT %QX."X20DO6639d".DigitalOutput01;
	Cyclic#2.::BrakeSetButton AT %IX."X20DI4653f".DigitalInput02;
	Cyclic#2.::MarkRFMoveOut AT %QX."X20DO6639d".DigitalOutput02;
	Cyclic#2.Brake8Inch2ndLeg AT %QX."X20DO6639e".DigitalOutput05;
	Cyclic#2.::MoveToBeam AT %QX."X20DO6639e".DigitalOutput01;
	Cyclic#2.::MoveAwayBeam AT %QX."X20DO6639e".DigitalOutput02;
END_VAR
```

## Configuration sim

CPU PC_any, AutomationRuntime J4.25, Build 4.1.2, Vc V4.25.0, Safety 0.0

### Task classes (Cpu.sw)
```
Cyclic#1 (cycle 10000 us, tolerance 10000 us):
  Server <- LibAsTCP1_ST.Server.prg
  MotionCont <- MotionControl1.prg
Cyclic#2 (cycle 20000 us, tolerance 50000000 us):
  Feeder <- Feeder.prg
  MarkTable <- MarkTable.prg
  MarkRF <- MarkRF.prg
  TDCTable <- TDCTable.prg
  TDCRFPshrs <- TDCRFPshrs.prg
  Insulmatic <- Insulmatic.prg
  GlueApp <- GlueApp.prg
  Pinspotter <- Pinspotter.prg
  BrakeCommo <- BrakeCommon.prg
  HWBwoPLC <- HWBwoPLC.prg
  HydraulicB <- HydraulicBrakeCarriage.prg
  CleatRoll <- CleatRoll.prg
Cyclic#4 (cycle 100000 us, tolerance 10000000 us):
  HMIButtons <- HMIButtons.prg
Cyclic#5 (cycle 2000000 us, tolerance 10000000 us):
  LampTest <- LampTest.prg
  Client <- LibAsTCP1_ST.Client.prg
Binaries: TCData, arconfig, asfw, ashwd, iomap, User, Role, sysconf
Libraries: standard, MestekLib, runtime, asieccon, astime, Library, asstring, astcp
```

### Hardware
```
PC : PC_any v1.1.0.0 (OrderNumber=PC)
  Connector IF1:
    ActivateDevice = 1
    ActivateIna = 1
  Connector IF3:
    InaPort = 11159
  ConfigurationID = X20_CPU_Config1
  Cyclic1Duration = 10000
  Cyclic1Tolerance = 10000
  Cyclic2Duration = 20000
  Cyclic2Tolerance = 50000000
  Cyclic3Duration = 50000
  Cyclic3Tolerance = 10000000
  Cyclic4Duration = 100000
  Cyclic4Tolerance = 10000000
  Cyclic5Duration = 2000000
  Cyclic5Tolerance = 10000000
  Cyclic6Duration = 3000000
  Cyclic6Tolerance = 12000000
  Cyclic7Duration = 4000000
  Cyclic7Tolerance = 12000000
  Cyclic8Duration = 5000000
  Cyclic8Tolerance = 30000000
```

## Logical view

Binary libraries used (declarations not repeated): operator, runtime, astime, AsIecCon, standard, AsTCP, asstring

### Global.var - Global variables
```iecst
VAR
	AccelRampReal : REAL := 500.0;
	AccelRampReal2 : REAL := 1000.0;
	ActlMetalEncoder : DINT;
	ActualDAC1 : INT;
	ActualDAC2 : INT;
	ActualMetalPosition : REAL; (*Scaled Material Position*)
	ActualRunPercent : REAL;
	ActualSpeed1 : REAL; (*Inches Per Second*)
	AdjustableTDCHeadActual : REAL;
	AdjustableTDCHeadDesired : REAL;
	AdjustableTDCHeadReference : REAL;
	AllSystemsOK : BOOL;
	AmberLight : BOOL;
	Analog1Forward : BOOL;
	Analog1Reverse : BOOL;
	AverageSpeed1 : REAL;
	BackGaugeAirBrake : BOOL;
	BackGaugeHomeLS : BOOL;
	BackGaugeJogInPB : BOOL;
	BackGaugeJogOutPB : BOOL;
	BackGaugeJogPercent : DINT;
	BackGaugeRunPercent : DINT;
	BatchActivePhysical : BOOL;
	BatchCancelSignal : BOOL;
	BC_Home4 : BOOL;
	BDelay1 : DINT;
	BDelay2 : DINT;
	BeadRollHits : DINT;
	BeadRollIndex : UINT;
	BeadRollJob : DINT;
	BeadRollMove : REAL;
	BeadRollTable : ARRAY[0..9] OF REAL;
	BeginEjectStep : BOOL;
	BeginMarkHoming : BOOL;
	BendingAgain : BOOL;
	BendingLatch : BOOL;
	BendInProcess : BOOL;
	BendSequenceReset : BOOL;
	BendStart : BOOL;
	BlockingValve : BOOL;
	BlockingValveButton : BOOL;
	BlueLight : BOOL;
	Brake8Inch2ndLeg : BOOL;
	BrakeActive : BOOL;
	BrakeActual : REAL := 20.0;
	BrakeArmLwrInhibit : BOOL;
	BrakeAuto : BOOL;
	BrakeAutoButton : BOOL;
	BrakeAutoIndicator : BOOL;
	BrakeAutoRequest : BOOL;
	BrakeBeamDownProx : BOOL;
	BrakeBeamLower : BOOL;
	BrakeBeamLwrInhibit : BOOL;
	BrakeBeamRaise : BOOL;
	BrakeBeamUpProx : BOOL;
	BrakeCarriageHomePosition : REAL;
	diBrakeCarriageJogIn : BOOL;
	diBrakeCarriageJogOut : BOOL;
	BrakeCarriageTarget : REAL;
	BrakeClampDownLS : BOOL;
	BrakeClampMidwayLS : BOOL;
	BrakeClampUpLS : BOOL;
	BrakeConveyorHigh : BOOL;
	BrakeConveyorLow : BOOL;
	BrakeDesired : REAL := 20.0;
	BrakeDriveEnable : BOOL;
	BrakeDriveFaultReset : BOOL;
	BrakeDriveReady : BOOL;
	BrakeDriveReset : BOOL;
	BrakeEncoder : DINT;
	BrakeEncoderReset : BOOL;
	BrakeHighSpeedRelay : BOOL;
	BrakeHiSpeedRelay : BOOL;
	BrakeHydraulicMS : BOOL;
	BrakeHydraulics : BOOL;
	BrakeIGain : DINT;
	BrakeInfeedConveyorMotor : BOOL;
	BrakeIsRefed : BOOL;
	BrakeIsSetUp : BOOL;
	BrakeJob : DINT;
	BrakeLeafHomeProx : BOOL;
	BrakeLeafLower : BOOL;
	BrakeLeafRaise : BOOL;
	BrakeLowSpeedRelay : BOOL;
	BrakeManualButton : BOOL;
	BrakeManualIndicator : BOOL;
	BrakeOn : BOOL;
	BrakeOutfeedConveyorMotor : BOOL;
	BrakePartEjectSolenoid : BOOL;
	BrakePartPresent : BOOL;
	BrakePercentSpeed : DINT;
	BrakePGain : DINT;
	BrakeReference : REAL;
	BrakeRefSignal : BOOL;
	BrakeRequired : BOOL;
	BrakeResolution : REAL;
	BrakeSequenceReset : BOOL;
	BrakeSetButton : BOOL;
	BrakeSingleCycle : BOOL;
	BrakeSlowWindow : DINT;
	BrakeSpeedSwitch : BOOL;
	BrakeStatus : DINT;
	BrakeStopsInSolenoid : BOOL;
	BrakeStopsOutSolenoid : BOOL;
	BrakeTarget0 : REAL;
	BrakeTarget1 : REAL;
	BrakeTarget2 : REAL;
	BrakeTarget3 : REAL;
	BrakeTargetWindow : DINT;
	BrakeTolerance : INT := 50; (*Servo*)
	ButtonActual : DINT;
	ButtonHits : DINT;
	ButtonIndex : USINT;
	ButtonJob : DINT;
	ButtonMove : REAL;
	ButtonRemainder : REAL;
	ButtonSignal : ARRAY[0..49] OF BOOL;
	ButtonStatus : ARRAY[0..49] OF BOOL;
	ButtonTable : ARRAY[0..5] OF REAL;
	BypassSwitch : BOOL;
	CaptureActl : ARRAY[0..49] OF DINT;
	CapturedAction : ARRAY[0..49] OF INT;
	CaptureIndex : INT;
	CaptureMetalTarget : ARRAY[0..49] OF DINT;
	CarriageArmLower : BOOL;
	CarriageArmRaise : BOOL;
	CarriageClampClose : BOOL;
	CarriageReference : BOOL;
	CDADecoilPower : BOOL;
	CEF1 : BOOL;
	CEF1Indicator : BOOL;
	CEF2 : BOOL;
	CEF2Indicator : BOOL;
	CEFJogPB : BOOL;
	CEFNotchDetect : BOOL;
	CEFPower : BOOL;
	CEFReset : BOOL;
	CenterDiePosition : ARRAY[0..17] OF BOOL;
	CenterHoleHits : DINT;
	CenterHoleIndex : USINT;
	CenterHoleMove : REAL;
	CenterHoleTable : ARRAY[0..17] OF REAL;
	CenterShuttleOutput : BOOL;
	ChangeBeadRoll : BOOL;
	ChangeConnector : BOOL;
	ChangeKDRolls : BOOL;
	CHoleDwell : DINT;
	CHoleJob : DINT;
	CHoleRemainder : REAL;
	CHoleValve : BOOL;
	CleanCycleLength : DINT;
	ClearLengthCountSignal : BOOL;
	CleatControl : DINT;
	CleatHits : DINT;
	CleatIndex : USINT;
	CleatJob : DINT;
	CleatMove : REAL;
	CleatOffDelay : DINT;
	CleatOnDelay : DINT;
	CleatRemainder : REAL;
	CleatRollerSheetSense : BOOL;
	CleatSide : DINT;
	CleatTable : ARRAY[0..5] OF REAL;
	CoilAccumulator : DINT;
	CoilLineHalt : BOOL;
	CoilLineHaltIndicator : BOOL;
	CoilLinePower : BOOL;
	CoilLineReset : BOOL;
	CoilLineRun : BOOL;
	CoilLineRunIndicator : BOOL;
	CoilLineSlowWindow : DINT;
	CoilLineTargetWindow : DINT;
	CoilWidth : REAL;
	ColdSealLeadDelay : DINT;
	ColdSealTrailDelay : DINT;
	ConfigureServos : BOOL;
	CropCut : BOOL;
	CropPercent1 : DINT;
	CushionRollRaiseSolenoid : BOOL;
	CustomLTDwell : DINT;
	CustomLTHits : DINT;
	CustomLTIndex : USINT;
	CustomLTJob : DINT;
	CustomLTMove : REAL;
	CustomLTRemainder : REAL;
	CustomLTTable : ARRAY[0..5] OF REAL;
	CustomLTValve : BOOL;
	CustomVDwell : DINT;
	CustomVHits : DINT;
	CustomVIndex : USINT;
	CustomVJob : DINT;
	CustomVMove : REAL;
	CustomVRemainder : REAL;
	CustomVTable : ARRAY[0..5] OF REAL;
	CustomVValve : BOOL;
	CycleButtons : BOOL;
	CycleCDie : BOOL;
	CycleCustomLTDie : BOOL;
	CycleCustomVDie : BOOL;
	CycleLDie : BOOL;
	CycleLTDie : BOOL;
	CycleMaleBender : BOOL;
	CycleRDie : BOOL;
	CycleShear : BOOL;
	CycleVDie : BOOL;
	DACAdd1 : REAL;
	DamperHoleSolenoid : BOOL;
	DClampTest : BOOL;
	DecelCounter : INT;
	DecelDistance1 : DINT;
	DecelRampReal : REAL := 500.0;
	DecelRampReal2 : REAL;
	DecelTime1 : REAL;
	DH800CEFCalibrateCR : BOOL;
	DH800CEFCalibratePB : BOOL;
	DH800CEFInCR : BOOL;
	DH800CEFInPB : BOOL;
	DH800CEFOutCR : BOOL;
	DH800CEFOutPB : BOOL;
	DH800CEFSlowCR : BOOL;
	DH800TInCR : BOOL;
	DH800TInPB : BOOL;
	DH800TOutCR : BOOL;
	DH800TOutPB : BOOL;
	diCoilSelectJog : BOOL;
	DieSelectSolenoid : BOOL;
	DieUpDelay : DINT;
	diFeedInitButton : BOOL;
	Difference : REAL;
	diMarkHeadDownProx : BOOL;
	diMarkHeadUpProx : BOOL;
	DischargeMarkSide : BOOL;
	DischargeTDCEnd : BOOL;
	DischargeTDCSide : BOOL;
	diTDCAdjustableHeadJogIn : BOOL;
	diTDCAdjustableHeadJogOut : BOOL;
	diTDCFixedHeadJogIn : BOOL;
	diTDCFixedHeadJogOut : BOOL;
	diTDCRollformerJog : BOOL;
	DLeafTest : BOOL;
	doCoilSelect : BOOL;
	doCoilSelectRollClose : BOOL;
	doMarkRFPassDown : BOOL;
	doMarkRFPassUp : BOOL;
	doMarkRollformerHeadLower : BOOL;
	doMarkRollformerHeadRaise : BOOL;
	DoneBending : BOOL;
	doProDuctHydraulics : BOOL;
	doTDCAdjustableHeadIn : BOOL;
	doTDCAdjustableHeadOut : BOOL;
	doTDCFixedHeadIn : BOOL;
	doTDCFixedHeadOut : BOOL;
	DuctoAuto : BOOL;
	DuctSelected : BOOL;
	DuctType : DINT;
	E1000CoilLine : BOOL;
	EjectComplete : BOOL;
	EjectPart1 : BOOL;
	ElectricDriveEnable : BOOL;
	ElectricDriveFaulted : BOOL;
	ElectricServoStuffOK : BOOL;
	ElectricWrapBrake : BOOL;
	EngelBrakeModelNumber : DINT;
	EngelCoilDriveReady : BOOL;
	EngelEServoOption : BOOL;
	EStopClear : BOOL;
	ExitBeltsOn : BOOL;
	EZPunchSolenoid : BOOL;
	FBBrakeSetSignal : BOOL;
	FeedInitButton : BOOL;
	FeedInitiate : BOOL;
	FirstTarget1 : BOOL;
	FittingDischargeType : DINT;
	FiveFootCenterSolenoid : BOOL;
	FiveFootOutsideSolenoid : BOOL;
	FixedTDCHeadActual : REAL;
	FixedTDCHeadDesired : REAL;
	FixedTDCHeadReference : REAL;
	FlushTubeRaiseTime : DINT;
	ForceBlockingValve : BOOL;
	FormHeadDownLS : BOOL;
	FormHeadDownSolenoid : BOOL;
	FormHeadUpLS : BOOL;
	FormHeadUpSolenoid : BOOL;
	ForwardFeedSolenoid : BOOL;
	FourFootCenterSolenoid : BOOL;
	FourFootOutsideSolenoid : BOOL;
	FSHydraulicsButton : BOOL;
	FullCleatButton : BOOL;
	FullCleatSelect : BOOL;
	FWBHome5 : BOOL;
	FWBResetPB : BOOL;
	FWBUnloaderValve : BOOL;
	GainsReceived : BOOL;
	GapTime : DINT;
	GChangeLShuttle : BOOL;
	GFeedMoveQed : BOOL;
	GLShuttleUnlatch : BOOL;
	GlueApplicatorType : DINT;
	GlueConveyorHiSpeedM : BOOL;
	GlueConveyorLowSpeedML : BOOL;
	GlueFlushPB : BOOL;
	GlueLeadDelay : DINT;
	GluePartSense : BOOL;
	GluePumpOnSwitch : BOOL;
	GlueServiceSwitch : BOOL;
	GlueSprayEnable : BOOL;
	GlueTrailDelay : DINT;
	GManualSignal : BOOL;
	GStep11 : BOOL;
	GStep12 : BOOL;
	GStep18 : BOOL;
	GStep18B : BOOL;
	GStep19 : BOOL;
	GStep21 : BOOL;
	GuideSideStopLS : BOOL;
	HasInsulmaticOnInput : BOOL;
	HeadInPositionLS : BOOL;
	HeartBeat : BOOL;
	HeavyIGain : DINT;
	HeavyPGain : DINT;
	hmiBrakeAutoButton : BOOL;
	hmiBrakeManualButton : BOOL;
	hmiFeedInitPB : BOOL;
	HolePunchSelectedSolenoid : BOOL;
	HolePunchUp : BOOL;
	HoleSize : BOOL;
	HumpLimitSwitch : BOOL;
	HWBCarriageInPosition : BOOL;
	HWBrakeWithNoPLC : BOOL;
	HWBrakeWithPLC : BOOL;
	ImaticBladeDown : BOOL;
	ImaticBladeUp : BOOL;
	ImaticFeedRoll : BOOL;
	ImaticPressRoll : BOOL;
	ImaticSquarePin : BOOL;
	IMotion2Target : DINT;
	IncrementalDINTTarget : DINT;
	IncrementalRealTarget : REAL;
	InCycle : BOOL;
	InPosition1 : BOOL;
	InPosition2 : BOOL;
	InsulationFeed : BOOL;
	InsulationRequired : BOOL;
	InsulmaticButton : BOOL;
	InsulmaticConveyorHi : BOOL;
	InsulmaticConveyorLow : BOOL;
	InsulmaticConveyorsOn : BOOL;
	InsulmaticEntranceHiSpeed : BOOL;
	InsulmaticEntranceLowSpeed : BOOL;
	InsulmaticExitHiSpeed : BOOL;
	InsulmaticExitLowSpeed : BOOL;
	InsulmaticLatch : BOOL;
	InsulmaticOn : BOOL;
	InsulmaticOnA : BOOL; (*Physical Input*)
	InsulmaticOnB : BOOL;
	InsulmaticSwingBlade : BOOL;
	InvalidDistREAL : REAL := -9999999.0;
	InvertShuttle : BOOL;
	ISquarePinOn : BOOL;
	ITmr1 : DINT;
	ITmr2 : DINT;
	ITmr3 : DINT;
	ITmr4 : DINT;
	ITmr5 : DINT;
	ITmr6 : DINT;
	ITmr7 : DINT;
	ITmr8 : DINT;
	ITmr9 : DINT;
	ITmr10 : DINT;
	ITmr11 : DINT;
	ITmr12 : DINT;
	ITmr13 : DINT;
	KnurledRollLength : REAL;
	LastPosition1 : DINT;
	LatchCylinderInLS : BOOL;
	LatchCylinderInSolenoid : BOOL;
	LatchCylinderOutLS : BOOL;
	LatchCylinderOutSolenoid : BOOL;
	LatestConnector : INT;
	LBrakeEjectorHomeProx : BOOL;
	LBrakeEjectorSwitch : BOOL;
	LBrakePartEjectSolenoid : BOOL;
	LBrakeWithNoPLC : BOOL;
	LBrakeWithPLC : BOOL;
	LBWN1 : BOOL;
	LBWN2 : BOOL;
	LBWN3 : BOOL;
	LBWN4 : BOOL;
	LBWN5 : BOOL;
	LBWN9 : BOOL;
	LBWN10 : BOOL;
	LBWN11 : BOOL;
	LBWNReady : BOOL;
	LeftCleatEnable : BOOL;
	LeftCleatKDRollValve : BOOL;
	LeftDiePosition : ARRAY[0..17] OF BOOL;
	LeftHoleHits : DINT;
	LeftHoleIndex : USINT;
	LeftHoleMove : REAL;
	LeftHoleTable : ARRAY[0..17] OF REAL;
	LeftKnockDownRoll : BOOL;
	LeftShuttleIndex : USINT;
	LeftShuttleOutput : BOOL;
	LevelerBrakeSolenoid : BOOL;
	LHoleDwell : DINT;
	LHoleJob : DINT;
	LHoleRemainder : REAL;
	LHoleValve : BOOL;
	Lift1Solenoid : BOOL;
	Lift2Solenoid : BOOL;
	Lift3DownDwell : TIME;
	Lift3DownProx : BOOL;
	Lift3DownSolenoid : BOOL;
	Lift3UpDwell : TIME;
	Lift3UpSolenoid : BOOL;
	LightIGain : DINT;
	LightPGain : DINT;
	LinerAirSupply : BOOL;
	LOMConveyorRunRelay : BOOL;
	LOMHiSpeedRelay : BOOL;
	LOMLowSpeedRelay : BOOL;
	LOMPower : BOOL;
	LOMSpeedSelect1 : BOOL;
	LOMSpeedSelect2 : BOOL;
	LTDwell : DINT;
	LTJob : DINT;
	LTNotchHits : DINT;
	LTNotchIndex : USINT;
	LTNotchMove : REAL;
	LTNotchTable : ARRAY[0..5] OF REAL;
	LTRemainder : REAL;
	LTValve : BOOL;
	MakeBeadRollTable : BOOL;
	MakeButtonTable : BOOL;
	MakeCHoleTable : BOOL;
	MakeCleatTable : BOOL;
	MakeCustomLTTable : BOOL;
	MakeCustomVTable : BOOL;
	MakeLHoleTable : BOOL;
	MakeLTTable : BOOL;
	MakeRHoleTable : BOOL;
	MakeShearBrakeTable : BOOL;
	MakeShearTable : BOOL;
	MakeVTable : BOOL;
	MaleLeafDwell : DINT;
	ManualClampPB : BOOL;
	Mark3PusherHome : BOOL;
	MarkActual : REAL;
	MarkAuto : BOOL;
	MarkButtonSignal : BOOL;
	MarkCleanDwell : DINT;
	MarkCleanLength : REAL;
	MarkConveyorDelayFwd : BOOL;
	MarkDesired : REAL;
END_VAR
VAR RETAIN
	MarkEncoder : DINT;
END_VAR
VAR
	MarkEncoderResetSignal : BOOL;
	MarkGateRaise : BOOL;
	MarkGateUpDwell : DINT;
	MarkHeadJoggingIn : BOOL;
	MarkHeadJoggingOut : BOOL;
	MarkHeadJogInSwitch : BOOL;
	MarkHeadJogOutSwitch : BOOL;
	MarkHiSpeedSignal : BOOL;
	MarkInPosBand : DINT;
	MarkMinLength : REAL;
	MarkPPauseDwell : DINT;
	MarkPshrFwd : BOOL;
	MarkPshrHome : BOOL;
	MarkPStageTime : DINT;
	MarkPStartDelay : DINT;
	MarkPStopDelay : DINT;
	MarkPushComplete : BOOL;
	MarkPusherReverse : BOOL;
	MarkPusherStop : BOOL;
	MarkReference : REAL;
	MarkRefSwitch : BOOL;
	MarkResolution : REAL;
END_VAR
VAR RETAIN
	MarkRFBase : DINT;
END_VAR
VAR
	MarkRFHighSpeed : BOOL;
	MarkRFInSignal : BOOL;
	MarkRFMoveIn : BOOL;
	MarkRFMoveOut : BOOL;
	MarkRFOutSignal : BOOL;
	MarkRollformerOn : BOOL;
	MarkSetButton : BOOL;
	MarkSetSignal : BOOL;
	MarkSlowBand : DINT;
	MarkStatus : DINT;
	MarkTableDecelDelay : DINT;
	MarkTableFwd : BOOL;
	MarkTableOn : BOOL;
	MarkTableRev : BOOL;
	MarkTableStart : BOOL;
	MarkTableStop : BOOL;
	MarkTarget : REAL;
	MarkTransferModel : DINT;
	MarkTTPusherJogRevPB : BOOL;
	MaterialClamped : BOOL;
	MatlAtMarkTable : BOOL;
	MatlAtMeasureRoll : BOOL;
	MaxCountsPerSecond : REAL;
	MaxDAC : INT := 32767;
	MaxDACSquared : REAL := 1073676289; (*Constant*)
	MaxRunJob : DINT := 500;
	MaxSpeed1 : REAL := 75.0; (*Feet Per Minute*)
	MediumIGain : DINT;
	MediumPGain : DINT;
	MetalActual : REAL;
	MetalDesired : REAL;
	MetalEncoder : DINT;
	MetalGauge : DINT;
	MetalScaler : REAL := 1.0;
	MetalTarget : DINT;
	MetalTolerance : INT := 30;
	MMCHeartBeat : BOOL;
	MotionStatus1 : INT := -1;
	MotionStatus2 : INT;
	MoveAwayBeam : BOOL;
	MoveCarriage : BOOL;
	MoveHeadRollSolenoid : BOOL;
	MoveMinus1 : BOOL;
	MoveMinus2 : BOOL;
	MoveMinus3 : BOOL;
	MovePlus1 : BOOL;
	MovePlus2 : BOOL;
	MovePlus3 : BOOL;
	MoveToBeam : BOOL;
	MTBlockedValve : BOOL;
	MTFlushTubeCloseSolenoid : BOOL;
	MTFlushTubeOpenSolenoid : BOOL;
	MTGlueValveSolenoid : BOOL;
	MTPlungerValveSolenoid : BOOL;
	MTWaterFlushSolenoid : BOOL;
	MTWaterSupplySolenoid : BOOL;
	NewRunJob : DINT;
	NextMoveDone : BOOL;
	NotchFFlag1 : DINT;
	NotchFFlag2 : DINT;
	NotchShuttleValve : BOOL;
	OneInchHolePunch : BOOL;
	OneMorePart : BOOL;
	OneSpeedExitBelts : BOOL;
	OperatorSideStopLS : BOOL;
	OutSideGuideSolenoid : BOOL;
	PartAtInsulationFeed : BOOL;
	PartAtISquarePin : BOOL;
	PartEjectHomeLS : BOOL;
	PartLength : REAL;
	PartPresentMarkExit : BOOL;
	PartPresentPSpotter : BOOL;
	PartPresentRTClamp : BOOL;
	PartPresentRTKnurledRoll : BOOL;
	PartRefOk : BOOL;
	PartRotateComplete : BOOL;
	PartsMade : DINT;
	PassThruButton : BOOL;
	PassThruPosition : BOOL;
	PCBrakeSetSignal : BOOL;
END_VAR
VAR RETAIN
	PercentJogSpeed1 : DINT := 10;
END_VAR
VAR
	PercentSpeed1 : DINT;
	PinDriveDwell : DINT;
	PinLoadDelay : DINT;
	PinLoadDwell : DINT;
	PinRepeat0 : DINT;
	PinRepeat1 : DINT;
	PinRepeat2 : DINT;
	PinRepeat3 : DINT;
	PinRepeat4 : DINT;
	PinRepeat5 : DINT;
	PinRepeat6 : DINT;
	PinRepeat7 : DINT;
	PinRepeat8 : DINT;
	PinRepeat9 : DINT;
	PinspotEncoder : DINT;
	PinspotEncoderResetSignal : BOOL;
	PinspotResolution : REAL;
	PinspotterDrive : BOOL;
	PinspotterLoad : BOOL;
	PinspotterSetSignal : BOOL;
	PinsRequired : BOOL;
	PinTarget0 : REAL;
	PinTarget1 : REAL;
	PinTarget2 : REAL;
	PinTarget3 : REAL;
	PinTarget4 : REAL;
	PinTarget5 : REAL;
	PinTarget6 : REAL;
	PinTarget7 : REAL;
	PinTarget8 : REAL;
	PinTarget9 : REAL;
	PittsButton : BOOL;
	PittsPosition : BOOL;
	PivotClampCloseSolenoid : BOOL;
	PivotClampLength : REAL;
	PivotTable : DINT;
	PivotTablePreset : ARRAY[0..12] OF TIME;
	PowerOn : BOOL;
	ProcessorDriveEnable : BOOL;
	ProcessorDriveReady : BOOL;
	ProcessorEncoderReset : BOOL;
	ProcessorJogFwd : BOOL;
	ProcessorJogRev : BOOL;
	PSpotActual : REAL;
	PSpotDesired : REAL;
	PunchMaster : BOOL;
	PunchMasterCoilWidth : REAL;
	PunchMasterShiftSolenoid : BOOL;
	PunchSelect : ARRAY[0..17] OF DINT;
	Pusher1OffProx : BOOL;
	Pusher1Solenoid : BOOL;
	Pusher2OffProx : BOOL;
	Pusher2Solenoid : BOOL;
	RaiseImaticBlade : BOOL;
	RaiseLeaf : BOOL;
	RaiseSquareArms : BOOL;
	RawMarkEncoder : DINT;
	RealBrakePosition : REAL;
	RealDAC1 : REAL;
	RearEjectResetLimitSwitch : BOOL;
	ReverseFeedSolenoid : BOOL;
	RHoleDwell : DINT;
	RHoleJob : DINT;
	RHoleRemainder : REAL;
	RHoleValve : BOOL;
	RightCleatEnable : BOOL;
	RightCleatKDRollValve : BOOL;
	RightDiePosition : ARRAY[0..17] OF BOOL;
	RightHoleHits : DINT;
	RightHoleIndex : USINT;
	RightHoleMove : REAL;
	RightHoleTable : ARRAY[0..17] OF REAL;
	RightKnockDownRoll : BOOL;
	RightShuttleIndex : INT;
	RightShuttleOutput : BOOL;
	RollDriveEnableButton : BOOL;
	RotateCompleteLength : REAL;
	RotateStopsOut : BOOL;
	RotatingTableOn : BOOL;
	RTBeltConveyorMotor : BOOL;
	RTBeltConveyorRaiseSolenoid : BOOL;
	RTKnurledRollGateSolenoid : BOOL;
	RTKnurledRollLowerSolenoid : BOOL;
	RTKnurledRollsMotor : BOOL;
	RTPivotArmRotate : BOOL;
	RTSkewTableRelay : BOOL;
	RunContinuousSignal : BOOL;
END_VAR
VAR RETAIN
	RunJob : DINT := 3;
END_VAR
VAR
	RunJobClick : BOOL;
	RunSpeed1 : DINT;
	SavedConnector : INT;
	SealantRequired : BOOL;
	SealantValve : BOOL;
	ServoLoop1Closed : BOOL;
	SetBendingSolenoids : BOOL;
	SettleTime1 : INT := 50;
	SettleTime2 : INT := 50;
	ShearBeamDownSS : BOOL;
	ShearBeamUpSS : BOOL;
	ShearBrakeHits : DINT;
	ShearBrakeIndex : USINT;
	ShearBrakeInstalled : BOOL;
	ShearBrakeJob : DINT;
	ShearBrakeLatch : BOOL;
	ShearBrakeMove : REAL;
	ShearBrakeReady : BOOL;
	ShearBrakeRemainder : REAL;
	ShearBrakeSetButton : BOOL;
	ShearBrakeTable : ARRAY[0..5] OF REAL;
	ShearClamp4Buttons : BOOL;
	ShearClampDownProx : BOOL;
	ShearClampLowerSolenoid : BOOL;
	ShearClampRaiseSolenoid : BOOL;
	ShearClampUpProx : BOOL;
	ShearDwell : DINT;
	ShearFFlag : DINT;
	ShearHits : DINT;
	ShearIndex : USINT;
	ShearJob : DINT;
	ShearLeafDownProx : BOOL;
	ShearLeafDownSS : BOOL;
	ShearLeafLowerSolenoid : BOOL;
	ShearLeafRaiseSolenoid : BOOL;
	ShearLeafUpProx : BOOL;
	ShearLeafUpSS : BOOL;
	ShearMove : REAL;
	ShearTable : ARRAY[0..5] OF REAL;
	ShearValve : BOOL;
	Short2ndLeg : BOOL;
	SideDischargeBrake : BOOL;
	SideEjectLiftSolenoid : BOOL;
	SideEjectSolenoid : BOOL;
	SixFootCenterSolenoid : BOOL;
	SixFootOutsideSolenoid : BOOL;
	SlackBar : BOOL;
	SlipAndDriveButton : BOOL;
	SlowSpeedSolenoid : BOOL;
	SmallPartPusherFwdSolenoid : BOOL;
	SmallPartPusherHomeLS : BOOL;
	SmallPartPusherRevSolenoid : BOOL;
	SmallPartsPusherLS : BOOL;
	SmallPittsSelected : BOOL;
	SnapButton : BOOL;
	SnapLockButtonGag : BOOL;
	SnapPosition : BOOL;
	SpareBool1 : BOOL;
	SpareBool2 : BOOL;
	SpareBool3 : BOOL;
	SpareBool4 : BOOL;
	SpareBool5 : BOOL;
	SRM1 : REAL;
	StandAloneCleatRoller : BOOL;
	StartSignal : BOOL;
	StartSignalClick : BOOL;
	StatHeadRollSolenoid : BOOL;
	Station1BrakeSolenoid : BOOL;
	Station1ForwardSolenoid : BOOL;
	Station1ReverseSolenoid : BOOL;
	Station2BrakeSolenoid : BOOL;
	Station2ForwardSolenoid : BOOL;
	Station2ReverseSolenoid : BOOL;
	Station3BrakeSolenoid : BOOL;
	Station3ReverseSolenoid : BOOL;
	Station4BrakeSolenoid : BOOL;
	Station4ForwardSolenoid : BOOL;
	Station4ReverseSolenoid : BOOL;
	Station5BrakeSolenoid : BOOL;
	Station5ForwardSolenoid : BOOL;
	Station5ReverseSolenoid : BOOL;
	Station6BrakeSolenoid : BOOL;
	Station6ForwardSolenoid : BOOL;
	Station6ReverseSolenoid : BOOL;
	Statrion3ForwardSolenoid : BOOL;
	Step01 : BOOL;
	Step02 : BOOL;
	Step03 : BOOL;
	Step04 : BOOL;
	Step04B : BOOL;
	Step04C : BOOL;
	Step04D : BOOL;
	Step04E : BOOL;
	Step08A : BOOL;
	Step08B : BOOL;
	Step13 : BOOL;
	Step14 : BOOL;
	StopFlag1 : BOOL;
	StopFlag2 : BOOL;
	StopWatch1 : REAL;
	Switch : BOOL;
	SystemHydraulicsOn : BOOL;
	Table1SheetStopProxA : BOOL;
	Table1SheetStopProxB : BOOL;
	Table1SideBypassLS : BOOL;
	Table2SheetStopProxA : BOOL;
	Table2SheetStopProxB : BOOL;
	TargetCount1 : INT;
	TargetDAC1 : INT;
	TDCAHeadPosition : DINT;
	TDCAutoWidthOption : BOOL;
	TDCConveyorRun : BOOL;
	TDCFixedHeadPosition : DINT;
	TDCHeadInPositionBand : REAL;
	TDCHeadReferenceButton : BOOL;
	TDCHeadReferenced : BOOL;
	TDCHeadResolution : REAL;
	TDCHeadSlowSpeedWindow : REAL;
	TDCHomePosition : REAL;
	TDCKnurlRollStyle : BOOL;
	TDCMotorLatch : BOOL;
	TDCNotchButton : BOOL;
	TDCPusherCycle : BOOL;
	TDCPusherEnable : BOOL;
	TDCPusherRevPB : BOOL;
	TDCPusherStyle : BOOL;
	TDCPushPartPresent : BOOL;
	TDCPushSetupDwell : DINT;
	TDCPushSignal : BOOL;
	TDCPushStrokeComplete : BOOL;
	TDCRFMotor : BOOL;
	TDCRFPushDelay : DINT;
	TDCRFPusherFwd : BOOL;
	TDCRFPusherIndicator : BOOL;
	TDCRFPusherRev : BOOL;
	TDCRFPusherStart : BOOL;
	TDCRFPusherStop : BOOL;
	TDCRFPusherStopDelay : DINT;
	TDCRunSignal : BOOL;
	TDCSetupOutputStyle : BOOL;
	TDCSquareDelay : DINT;
	TDCTableLength : REAL;
	TDCTableOn : BOOL;
	TDCTablePartProx : BOOL;
	TDCTablePause : BOOL;
	TDCTablePauseDwell : DINT;
	TDCTablePusherFwd : BOOL;
	TDCTablePusherReverse : BOOL;
	TDCTablePusherRevPB : BOOL;
	TDCTablePushStop : BOOL;
	TDCTableStop : BOOL;
	TDCTransferOnIndicator : BOOL;
	TDCTransferTableButton : BOOL;
	TDCTTLatch : BOOL;
	TDFJogPB : BOOL;
	TDFPower : BOOL;
	TopDAC1 : INT;
	TopLineSpeed : REAL; (*Inches Per Second*)
	TotalInches : REAL := 864;
	Transfer1Power : BOOL;
	Transfer2Power : BOOL;
	TransferSystemPower : BOOL;
	TripIndicatorBrake : BOOL;
	TripIndicatorCEF : BOOL;
	TripIndicatorCoilLine : BOOL;
	TripIndicatorCradles2 : BOOL;
	TripIndicatorPump : BOOL;
	TripIndicatorTDF : BOOL;
	TripIndicatorTransfer1 : BOOL;
	TripIndicatorTransfer2 : BOOL;
	TSBrakeDriveResetButton : BOOL;
	TSBrakeHydraulicsButton : BOOL;
	TSCDAButton : BOOL;
	TSCEF1Button : BOOL;
	TSCEF2Button : BOOL;
	TSCEFButton : BOOL;
	TSLOMButton : BOOL;
	TSTDFButton : BOOL;
	TSTransferButton : BOOL;
	UClampTest : BOOL;
	ULeafTest : BOOL;
	ULineSelected : BOOL;
	Uncoiler1Select : BOOL;
	Uncoiler2Select : BOOL;
	Uncoiler3Select : BOOL;
	Uncoiler4Select : BOOL;
	Uncoiler5Select : BOOL;
	Uncoiler6Select : BOOL;
	UncoilerAutoSwitch : BOOL;
	UncoilerForwardSolenoid : BOOL;
	UncoilerJogForwardPB : BOOL;
	UncoilerJogForwardPB_A : BOOL;
	UncoilerJogPB : BOOL;
	UncoilerJogReversePB : BOOL;
	UncoilerLoad : BOOL;
	UncoilerOnLatch : BOOL;
	UncoilerReverseSolenoid : BOOL;
	UncoilerRewindSwitch : BOOL;
	UncoilerRun : BOOL;
	UncoilerRunA : BOOL;
	UncoilerRunB : BOOL;
	UncoilerRunMode : BOOL;
	UncoilerStationLimitSwitch1 : BOOL;
	UncoilerStationLimitSwitch2 : BOOL;
	UncoilerStationLimitSwitch3 : BOOL;
	UncoilerStationLimitSwitch4 : BOOL;
	UncoilerStationLimitSwitch5 : BOOL;
	UncoilerStationLimitSwitch6 : BOOL;
	UncoilerUnwindSwitch : BOOL;
	UnitsPerInch1 : REAL := 2000.0;
	UpdateRate1 : INT := 1;
	UpdateRate2 : USINT := 1;
	UpdateTablesDone : BOOL;
	VDwell : DINT;
	VJob : DINT;
	VNotchHits : DINT;
	VNotchIndex : USINT;
	VNotchMove : REAL;
	VNotchTable : ARRAY[0..5] OF REAL;
	VRemainder : REAL;
	VValve : BOOL;
	WaitCon3 : BOOL;
	WaitToFire1 : BOOL;
	WaitToFire2 : BOOL;
	WaitToFire3 : BOOL;
	WarningComplete : BOOL;
	WarningDelay1 : TIME := T#10ms;
	WarningHorn : BOOL;
	WB1BendDoneStep : BOOL;
	WBArmsUpStep : BOOL;
	WBAutoStep : BOOL;
	WBBendingStep : BOOL;
	WBBendSeqStartStep : BOOL;
	WBBrakeRequiredStep : BOOL;
	WBCarriageReturningStep : BOOL;
	WBCarriageReturnStep : BOOL;
	WBCloseClampStep : BOOL;
	WBLowerCarriageArmsStep : BOOL;
	WBMachineSetStep : BOOL;
	WBNotClampedStep : BOOL;
	WBNotInPositionStep : BOOL;
	WBOpenClampStep : BOOL;
	WBPartPastStep : BOOL;
	WBPartPresentStep : BOOL;
	WBPreset1 : TIME;
	WBPreset2 : TIME;
	WBPreset3 : TIME;
	WBPreset4 : TIME;
	WBPreset5 : TIME;
	WBPreset6 : TIME;
	WBRaiseArmsStep : BOOL;
	WBRaiseLeafStep : BOOL;
	diWBrakeArmsUp : BOOL;
	WBReadyToCycleStep : BOOL;
	WBSequenceComplete : BOOL;
	WBSquareStep : BOOL;
	ZeroCropButton : BOOL;
	ZeroCropCut : BOOL;
	ZeroCropOffset : REAL;
	WBMissedPart : BOOL;
	BrakeEjectTarget : REAL;
	IBrakeReference : DINT;
	Block_1 : BOOL;
END_VAR
```

### Package Logical/Libraries - Global libraries

### Library Logical/Libraries/MestekLib (IEC)

#### MestekLib.fun - Exported functions and function blocks
```iecst
FUNCTION myAdd : REAL (*Adds two numbers together*) (*$GROUP=User,$CAT=User,$GROUPICON=User.png,$CATICON=User.png*)
	VAR_INPUT
		val1 : REAL;
		val2 : REAL;
	END_VAR
END_FUNCTION
```

#### myAdd.st
```iecst
(* Adds two numbers together *)
FUNCTION myAdd

	myAdd	:= val1 + val2;

END_FUNCTION
```

### Program Logical/LampTest (IEC)

#### Variables.var
```iecst
VAR
	Lamp : BOOL;
END_VAR
```

#### Cyclic.ld
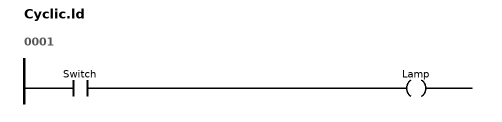
Ladder, written as Structured Text:
```iecst
PROGRAM _CYCLIC
(* Network 1 *)
Lamp := Switch;
END_PROGRAM
```

### Program Logical/MotionControl1 (IEC)

#### Cyclic.st
```iecst
PROGRAM _CYCLIC
	difference := MetalTarget - ActlMetalEncoder;
	AbsoluteDifference := ABS(difference);
	CASE MotionStatus1 OF
		(*Hold Position*)
		0:
			IF NOT InPosition1 THEN
				IF AbsoluteDifference <= MetalTolerance THEN
					TargetCount1 := TargetCount1 + UpdateRate1;
					IF TargetCount1 >= SettleTime1 THEN
						InPosition1 := TRUE;
					END_IF;
				END_IF;
			END_IF;

			Ratio1 := DINT_TO_INT(difference + (difference / 2));
			IF Counter1 > 0 THEN
				Counter1 := Counter1 - UpdateRate1;
			ELSE
				Counter1 := 500;
				IF Hold1 <> Ratio1 THEN
					Hold1 := Ratio1;
				ELSE
					DACBalance1 := ActualDAC1;
				END_IF;
			END_IF;

			TargetDAC1 := Ratio1 + DACBalance1;
			IF TargetDAC1 >= ActualDAC1 THEN
				IF TargetDAC1 - ActualDAC1 > (10 * UpdateRate1) THEN
					ActualDAC1 := ActualDAC1 + (10 * UpdateRate1);
				ELSE
					ActualDAC1 := TargetDAC1;
				END_IF;
			ELSE
				IF ActualDAC1 - TargetDAC1 > (10 * UpdateRate1) THEN
					ActualDAC1 := ActualDAC1 - (10 * UpdateRate1);
				ELSE
					ActualDAC1 := TargetDAC1;
				END_IF;
			END_IF;

			IF ActualDAC1 > TopDAC1 THEN
				ActualDAC1 := TopDAC1;
			END_IF;
			IF ActualDAC1 < -TopDAC1 THEN
				ActualDAC1 := -TopDAC1;
			END_IF

		(*Initialize Move*)
		1:
			CoilAccumulator := MetalTarget; (*Update Accumulator to last target*)
			(*IncrementalRealTarget is the amount required to move determined elsewhere*)
			IncrementalDINTTarget := REAL_TO_DINT(IncrementalRealTarget * UnitsPerInch1 * MetalScaler);
			MetalTarget := MetalTarget + IncrementalDINTTarget;
			TopDAC1 := DINT_TO_INT((INT_TO_DINT(MaxDAC) * RunSpeed1) / 100);
			ActualSpeed1 := ((MaxSpeed1 / 5.0) * DINT_TO_REAL(RunSpeed1)) / 100.0; (*Real Inches Per Second*)
			AverageSpeed1 := ActualSpeed1 / 2.0;
			DecelTime1 := (DecelRampReal / 1000.0) * (DINT_TO_REAL(RunSpeed1) / 100);
			DecelDistance1 := REAL_TO_DINT(((AverageSpeed1 * DecelTime1) * MetalScaler) * UnitsPerInch1);
			MaxCountsPerSecond := (MaxSpeed1 / 5.0) * UnitsPerInch1;
			SRM1 := MaxDACSquared / ((MaxCountsPerSecond * (DecelRampReal / 1000.0)) / 2.0);
			IF DecelDistance1 > IncrementalDINTTarget THEN
				DecelDistance1 := IncrementalDINTTarget / 2;
				TopDAC1 := REAL_TO_INT(SQRT(DINT_TO_REAL(DecelDistance1) / MetalScaler) * SRM1);
				IF TopDAC1 < 50 THEN
					TopDAC1 := 50;
				END_IF;
			END_IF;
			InPosition1 := FALSE;
			FirstTarget1 := FALSE;
			StopWatch1 := 0.0;
			DACAdd1 := INT_TO_REAL(MaxDAC) / AccelRampReal;
			MotionStatus1 := 2;
		(*Ramp Up To Speed*)
		2:
			IF DecelDistance1 < difference THEN
				IF ActualDAC1 < TopDAC1 THEN (*Accelerate*)
					StopWatch1 := StopWatch1 + INT_TO_REAL(UpdateRate1);
					ActualDAC1 := REAL_TO_INT(StopWatch1 * DACAdd1);
				ELSE  (*Constant Speed*)
					ActualDAC1 := TopDAC1;
				END_IF;
			ELSE (*Switch To Decel MotionState*)
				DecelCounter := 25;
				LastPosition1 := ActlMetalEncoder;
				TargetCount1 := 0;
				FirstTarget1 := FALSE;
				MotionStatus1 := 3;
			END_IF;
		3:
			(*Stall Detection*)
			DecelCounter := DecelCounter - UpdateRate1;
			IF DecelCounter = 0 THEN
				DecelCounter := 100;
				IF LastPosition1 = ActualMetalPosition THEN
					TopDAC1 := MaxDAC / 4;
					MotionStatus1 := 0;
				ELSE
					LastPosition1 := ActlMetalEncoder;
				END_IF;
			END_IF;

			ActualDAC1 := REAL_TO_INT(DINT_TO_REAL(AbsoluteDifference) * SRM1);

			IF difference < 0 THEN
				ActualDAC1 := -ActualDAC1;
			END_IF;

			IF FirstTarget1 THEN
				ActualDAC1 := ActualDAC1 / 8;
			END_IF;

			IF AbsoluteDifference < MetalTolerance THEN
				FirstTarget1 := TRUE;
				TargetCount1 := TargetCount1 + UpdateRate1;
				IF TargetCount1 >= SettleTime1 THEN
					InPosition1 := TRUE;
					MotionStatus1 := 0;
					TopDAC1 := MaxDAC / 4;
				END_IF;
			ELSE
				TargetCount1 := 0;
			END_IF;
		4: (*Setup Forward Jog*)
			DACAdd1 := INT_TO_REAL(MaxDAC) / AccelRampReal;
			TopDAC1 := DINT_TO_INT((INT_TO_DINT(MaxDAC) * PercentJogSpeed1) / 100);
			StopFlag1 := FALSE;
			MotionStatus1 := 7;
		5: (*Setup Reverse Jog*)
			DACAdd1 := INT_TO_REAL(MaxDAC) / AccelRampReal;
			TopDAC1 := DINT_TO_INT((INT_TO_DINT(MaxDAC) * PercentJogSpeed1) / 100);
			StopFlag1 := FALSE;
			MotionStatus1 := 8;
		7: (*Forward Jog*)
			IF StopFlag1 THEN
				IF ActualDAC1 > REAL_TO_INT(DACAdd1) THEN (*Decelerate*)
					ActualDAC1 := ActualDAC1 - REAL_TO_INT(DACAdd1);
				ELSE (*Hold Position*)
					ActualDAC1 := 0;
					MetalTarget := ActlMetalEncoder;
					MotionStatus1 := -1;
				END_IF;
			ELSE
				IF ActualDAC1 < TopDAC1 THEN (*Accelerate*)
					ActualDAC1 := ActualDAC1 + REAL_TO_INT(DACAdd1);
				ELSE
					ActualDAC1 := TopDAC1; (*Maintain Constant Speed*)
				END_IF;
			END_IF;
		8: (*Reverse Jog*)
			IF StopFlag1 THEN
				IF ActualDAC1 < REAL_TO_INT(-DACAdd1) THEN (*Decelerate*)
					ActualDAC1 := ActualDAC1 + REAL_TO_INT(DACAdd1);
				ELSE (*Hold Position*)
					ActualDAC1 := 0;
					MetalTarget := ActlMetalEncoder;
					MotionStatus1 := -1;
				END_IF;
			ELSE
				IF ActualDAC1 > -TopDAC1 THEN (*Accelerate*)
					ActualDAC1 := ActualDAC1 - REAL_TO_INT(DACAdd1);
				ELSE
					ActualDAC1 := TopDAC1; (*Maintain Constant Speed*)
				END_IF;
			END_IF;
		ELSE (*Not Moving Or Holding*)
		  ActualDAC1 := 0;
		  MetalTarget := ActlMetalEncoder;
		  InPosition1 := TRUE;
	END_CASE;

	IF ActualDAC1 > MaxDAC THEN
		ActualDAC1 := MaxDAC;
	END_IF;
	IF ActualDAC1 < -MaxDAC THEN
		ActualDAC1 := -MaxDAC;
	END_IF;

END_PROGRAM
```
